# B&R Automation Studio project NAEUL004C00R13L518F00 (part 60)

#### InputRef.var - not listed in the package file held
```iecst
(*2019-03-22*)
(**)
(*General*)
VAR
	p_udiMax : REFERENCE TO UDINT;
	p_udiRstErr : REFERENCE TO UDINT;
END_VAR
(**)
(*Configuration*)
VAR
	p_tyDISettings : REFERENCE TO tyDigitalInputSettings;
	p_sProgNm : REFERENCE TO STRING[15];
END_VAR
(**)
VAR
	p_diConvLftSenOnTm : REFERENCE TO DINT;
	p_diConvLftSenOffTm : REFERENCE TO DINT;
	p_diConvMidSenOnTm : REFERENCE TO DINT;
	p_diConvMidSenOffTm : REFERENCE TO DINT;
	p_diConvRgtSenOnTm : REFERENCE TO DINT;
	p_diConvRgtSenOffTm : REFERENCE TO DINT;
	p_diConvClrSenOnTm : REFERENCE TO DINT;
	p_diConvClrSenOffTm : REFERENCE TO DINT;
	p_diMagConvEntSenOnTm : REFERENCE TO DINT;
	p_diMagConvEntSenOffTm : REFERENCE TO DINT;
	p_diMagConvPresentSenOnTm : REFERENCE TO DINT;
	p_diMagConvPresentSenOffTm : REFERENCE TO DINT;
	p_diConvLineAInletSenOnTm : REFERENCE TO DINT;
	p_diConvLineAInletSenOffTm : REFERENCE TO DINT;
	p_diConvLineBInletSenOnTm : REFERENCE TO DINT;
	p_diConvLineBInletSenOffTm : REFERENCE TO DINT;
	p_diConvUSWidthChkSenOnTm : REFERENCE TO DINT;
	p_diConvUSWidthChkSenOffTm : REFERENCE TO DINT;
	p_tyNtParamCurr : REFERENCE TO tyNtParam;
	p_bMcParamUSWidthChkEn : REFERENCE TO BOOL;
END_VAR
(*Self Test Var*)
VAR
	p_bSelfTest : REFERENCE TO BOOL;
	p_bPshrConvHvBrd : REFERENCE TO BOOL;
	p_tyBufferStat1 : REFERENCE TO tyBffrStat;
	p_tyBufferStat2 : REFERENCE TO tyBffrStat;
	p_tyBufferStat3 : REFERENCE TO tyBffrStat;
	p_tySOTSimulate1 : REFERENCE TO tySOTSigmulateSig;
	p_tySOTSimulate2 : REFERENCE TO tySOTSigmulateSig;
	p_tySOTSimulate3 : REFERENCE TO tySOTSigmulateSig;
	p_bUIAGVSimulationOn : REFERENCE TO BOOL;
	p_tyTagFromMes : REFERENCE TO tyStatFromMES;
	p_tyDO : REFERENCE TO tyDigitalOutput;
	p_eULMag : REFERENCE TO eULMag;
	p_bRstErrSafetyRlyRst : REFERENCE TO BOOL;
	p_bRstCurtainSen : REFERENCE TO BOOL;
END_VAR
(*MagConv On/Off Tm*)
VAR
	p_diInMagConvEntSenOnTm : REFERENCE TO DINT;
	p_diInMagConvEntSenOffTm : REFERENCE TO DINT;
	p_diInMagConvExtSenOnTm : REFERENCE TO DINT;
	p_diInMagConvExtSenOffTm : REFERENCE TO DINT;
	p_diInMagConvMidSenOnTm : REFERENCE TO DINT;
	p_diInMagConvMidSenOffTm : REFERENCE TO DINT;
	p_diOutMagConvEntSenOnTm : REFERENCE TO DINT;
	p_diOutMagConvEntSenOffTm : REFERENCE TO DINT;
	p_diOutMagConvExtSenOnTm : REFERENCE TO DINT;
	p_diOutMagConvExtSenOffTm : REFERENCE TO DINT;
	p_diOutMagConvMidSenOnTm : REFERENCE TO DINT;
	p_diOutMagConvMidSenOffTm : REFERENCE TO DINT;
	p_diInMagConv2EntSenOnTm : REFERENCE TO DINT;
	p_diInMagConv2EntSenOffTm : REFERENCE TO DINT;
	p_diInMagConv2ExtSenOnTm : REFERENCE TO DINT;
	p_diInMagConv2ExtSenOffTm : REFERENCE TO DINT;
	p_diInMagConv2MidSenOnTm : REFERENCE TO DINT;
	p_diInMagConv2MidSenOffTm : REFERENCE TO DINT;
	p_diOutMagConv2EntSenOnTm : REFERENCE TO DINT;
	p_diOutMagConv2EntSenOffTm : REFERENCE TO DINT;
	p_diOutMagConv2ExtSenOnTm : REFERENCE TO DINT;
	p_diOutMagConv2ExtSenOffTm : REFERENCE TO DINT;
	p_diOutMagConv2MidSenOnTm : REFERENCE TO DINT;
	p_diOutMagConv2MidSenOffTm : REFERENCE TO DINT;
	p_bOpsRun : REFERENCE TO BOOL;
	p_bManual : REFERENCE TO BOOL;
	p_bCurtainSenPrep : REFERENCE TO BOOL;
	p_bBypassLifMagInletShute : REFERENCE TO BOOL;
	p_eMidSenNcNoType : REFERENCE TO eMidSenParam;
END_VAR
```

#### InputRef_Link.var - not listed in the package file held
```iecst
(*2019-04-09*)
(**)
(*External Data*)
VAR
	p_eLinkAGVComProtocol : REFERENCE TO eMcAGVCommProtocol;
	p_bLinkNtParamProjSOTSenPrep : REFERENCE TO BOOL;
	p_bLinkStartupRun : REFERENCE TO BOOL;
	p_bOpsTravLifULBypCurtainSenCtrl : REFERENCE TO BOOL;
END_VAR
```

#### Act_Alarm1.st - not listed in the package file held
```iecst
(** 2019-03-25 **)
ACTION Act_Alarm1:

	//Error
	IF EDGEPOS(eStatus1 = Error) THEN

		tyAlmData1.sProgNm		:= p_sProgNm;
		tyAlmData1.udiCode		:= udiStatus1;
		tyAlmData1.eSeverity	:= AlmSeverityError;
		tyAlmData1.udiRunTime	:= tyAlmData1.udiRunTime + 1;
		tyAlmData1.bAlm			:= TRUE;
		tyAlmData1.udiModuleNum  := udiModuleNum;
		g_sDInputProgNm		:= p_sProgNm;

		//Get Error Message
		IF tyAlmData1.udiCode < 10000 OR tyAlmData1.udiCode > 10099 THEN
			tyAlmData1.sAlmMsg	:= 'Unknown';
			tyAlmData1.sRcyMsg	:= 'Unknown';
		ELSE
			tyAlmData1.sAlmMsg	:= a_tyAlmText[tyAlmData1.udiCode].sAlmText;
			tyAlmData1.sRcyMsg	:= a_tyAlmText[tyAlmData1.udiCode].sRcyText;
		END_IF

	ELSIF bRstErr AND (tyAlmData1.udiCode <> 0) THEN

		tyAlmData1.udiCode		:= 0;
		tyAlmData1.eSeverity	:= AlmSeverityNA;
		tyAlmData1.sAlmMsg		:= '';
		tyAlmData1.sRcyMsg		:= '';
		tyAlmData1.bAlm			:= FALSE;
	END_IF

END_ACTION
```

#### Act_Alarm2.st - not listed in the package file held
```iecst
(** 2019-03-25 **)
ACTION Act_Alarm2:

	//Error
	IF EDGEPOS(eStatus2 = Error) THEN

		tyAlmData2.sProgNm		:= p_sProgNm;
		tyAlmData2.udiCode		:= udiStatus2;
		tyAlmData2.eSeverity	:= AlmSeverityError;
		tyAlmData2.udiRunTime	:= tyAlmData2.udiRunTime + 1;
		tyAlmData2.bAlm			:= TRUE;
		tyAlmData2.udiModuleNum  := udiModuleNum;
		g_sDInputProgNm		:= p_sProgNm;
		//Get Error Message
		IF tyAlmData2.udiCode < 10000 OR tyAlmData2.udiCode > 10099 THEN
			tyAlmData2.sAlmMsg	:= 'Unknown';
			tyAlmData2.sRcyMsg	:= 'Unknown';
		ELSE
			tyAlmData2.sAlmMsg	:= a_tyAlmText[tyAlmData2.udiCode].sAlmText;
			tyAlmData2.sRcyMsg	:= a_tyAlmText[tyAlmData2.udiCode].sRcyText;
		END_IF

	ELSIF bRstErr AND (tyAlmData2.udiCode <> 0) THEN

		tyAlmData2.udiCode		:= 0;
		tyAlmData2.eSeverity	:= AlmSeverityNA;
		tyAlmData2.sAlmMsg		:= '';
		tyAlmData2.sRcyMsg		:= '';
		tyAlmData2.bAlm			:= FALSE;
	END_IF

END_ACTION
```

#### Act_Alarm3.st - not listed in the package file held
```iecst
(** 2019-03-25 **)
ACTION Act_Alarm3:

	//Error
	IF EDGEPOS(eStatus3 = Error) THEN

		tyAlmData3.sProgNm		:= p_sProgNm;
		tyAlmData3.udiCode		:= udiStatus3;
		tyAlmData3.eSeverity	:= AlmSeverityError;
		tyAlmData3.udiRunTime	:= tyAlmData3.udiRunTime + 1;
		tyAlmData3.bAlm			:= TRUE;
		tyAlmData3.udiModuleNum  := udiModuleNum;
		g_sDInputProgNm		:= p_sProgNm;
		//Get Error Message
		IF tyAlmData3.udiCode < 10000 OR tyAlmData3.udiCode > 10099 THEN
			tyAlmData3.sAlmMsg	:= 'Unknown';
			tyAlmData3.sRcyMsg	:= 'Unknown';
		ELSE
			tyAlmData3.sAlmMsg	:= a_tyAlmText[tyAlmData3.udiCode].sAlmText;
			tyAlmData3.sRcyMsg	:= a_tyAlmText[tyAlmData3.udiCode].sRcyText;
		END_IF

	ELSIF bRstErr AND (tyAlmData3.udiCode <> 0) THEN

		tyAlmData3.udiCode		:= 0;
		tyAlmData3.eSeverity	:= AlmSeverityNA;
		tyAlmData3.sAlmMsg		:= '';
		tyAlmData3.sRcyMsg		:= '';
		tyAlmData3.bAlm			:= FALSE;
	END_IF

END_ACTION
```

#### Act_Alarm4.st - not listed in the package file held
```iecst
(** 2019-03-25 **)
ACTION Act_Alarm4:

	//Error
	IF EDGEPOS(eStatus4 = Error) THEN

		tyAlmData4.sProgNm		:= p_sProgNm;
		tyAlmData4.udiCode		:= udiStatus4;
		tyAlmData4.eSeverity	:= AlmSeverityError;
		tyAlmData4.udiRunTime	:= tyAlmData4.udiRunTime + 1;
		tyAlmData4.bAlm			:= TRUE;
		tyAlmData4.udiModuleNum  := udiModuleNum;
		g_sDInputProgNm		:= p_sProgNm;
		//Get Error Message
		IF tyAlmData4.udiCode < 10000 OR tyAlmData4.udiCode > 10099 THEN
			tyAlmData4.sAlmMsg	:= 'Unknown';
			tyAlmData4.sRcyMsg	:= 'Unknown';
		ELSE
			tyAlmData4.sAlmMsg	:= a_tyAlmText[tyAlmData4.udiCode].sAlmText;
			tyAlmData4.sRcyMsg	:= a_tyAlmText[tyAlmData4.udiCode].sRcyText;
		END_IF

	ELSIF bRstErr AND (tyAlmData4.udiCode <> 0) THEN

		tyAlmData4.udiCode		:= 0;
		tyAlmData4.eSeverity	:= AlmSeverityNA;
		tyAlmData4.sAlmMsg		:= '';
		tyAlmData4.sRcyMsg		:= '';
		tyAlmData4.bAlm			:= FALSE;
	END_IF

END_ACTION
```

#### Act_Alarm5.st - not listed in the package file held
```iecst
(** 2019-03-25 **)
ACTION Act_Alarm5:

	//Error
	IF EDGEPOS(eStatus5 = Error) THEN

		tyAlmData5.sProgNm		:= p_sProgNm;
		tyAlmData5.udiCode		:= udiStatus5;
		tyAlmData5.eSeverity	:= AlmSeverityError;
		tyAlmData5.udiRunTime	:= tyAlmData5.udiRunTime + 1;
		tyAlmData5.bAlm			:= TRUE;
		tyAlmData5.udiModuleNum  := udiModuleNum;
		g_sDInputProgNm		:= p_sProgNm;
		//Get Error Message
		IF tyAlmData5.udiCode < 10000 OR tyAlmData5.udiCode > 10099 THEN
			tyAlmData5.sAlmMsg	:= 'Unknown';
			tyAlmData5.sRcyMsg	:= 'Unknown';
		ELSE
			tyAlmData5.sAlmMsg	:= a_tyAlmText[tyAlmData5.udiCode].sAlmText;
			tyAlmData5.sRcyMsg	:= a_tyAlmText[tyAlmData5.udiCode].sRcyText;
		END_IF

	ELSIF bRstErr AND (tyAlmData5.udiCode <> 0) THEN

		tyAlmData5.udiCode		:= 0;
		tyAlmData5.eSeverity	:= AlmSeverityNA;
		tyAlmData5.sAlmMsg		:= '';
		tyAlmData5.sRcyMsg		:= '';
		tyAlmData5.bAlm			:= FALSE;
	END_IF

END_ACTION
```

#### Act_Alarm6.st - not listed in the package file held
```iecst
(** 2019-03-25 **)
ACTION Act_Alarm6:

	//Error
	IF EDGEPOS(eStatus6 = Error) THEN

		tyAlmData6.sProgNm		:= p_sProgNm;
		tyAlmData6.udiCode		:= udiStatus6;
		tyAlmData6.eSeverity	:= AlmSeverityError;
		tyAlmData6.udiRunTime	:= tyAlmData6.udiRunTime + 1;
		tyAlmData6.bAlm			:= TRUE;
		tyAlmData6.udiModuleNum  := udiModuleNum;
		g_sDInputProgNm		:= p_sProgNm;
		//Get Error Message
		IF tyAlmData6.udiCode < 10000 OR tyAlmData6.udiCode > 10099 THEN
			tyAlmData6.sAlmMsg	:= 'Unknown';
			tyAlmData6.sRcyMsg	:= 'Unknown';
		ELSE
			tyAlmData6.sAlmMsg	:= a_tyAlmText[tyAlmData6.udiCode].sAlmText;
			tyAlmData6.sRcyMsg	:= a_tyAlmText[tyAlmData6.udiCode].sRcyText;
		END_IF

	ELSIF bRstErr AND (tyAlmData6.udiCode <> 0) THEN

		tyAlmData6.udiCode		:= 0;
		tyAlmData6.eSeverity	:= AlmSeverityNA;
		tyAlmData6.sAlmMsg		:= '';
		tyAlmData6.sRcyMsg		:= '';
		tyAlmData6.bAlm			:= FALSE;
	END_IF

END_ACTION
```

#### Act_InitGlobal.st - not listed in the package file held
```iecst
(** 2018-12-10 **)
ACTION Act_InitGlobal:

	(* Always Change If Project Change *)

	//Pass Data To Link
	p_eLinkAGVComProtocol ACCESS p_McParamAGVComProtocol;
	p_bLinkNtParamProjSOTSenPrep ACCESS p_NtParamProjSOTSenPrep;
	p_bLinkStartupRun ACCESS p_StartupRun;
	p_bOpsTravLifULBypCurtainSenCtrl ACCESS p_OpsTravLifULBypCurtainSenCtrl;
	p_bOpsRun ACCESS p_OpsRun;
	p_bCurtainSenPrep ACCESS p_NtParamCurtainSenPrep;

	//Pass Data To Internal Use
	p_udiRstErr ACCESS p_RstErrReset;
	p_tyDISettings ACCESS p_NtParamDISettings;
	p_sProgNm ACCESS p_NtParamDIProgNm;

	p_diConvLftSenOnTm ACCESS p_McParamConvLftSenOnTm;
	p_diConvLftSenOffTm ACCESS p_McParamConvLftSenOffTm;
	p_diConvMidSenOnTm ACCESS p_McParamConvMidSenOnTm;
	p_diConvMidSenOffTm ACCESS p_McParamConvMidSenOffTm;
	p_diConvRgtSenOnTm ACCESS p_McParamConvRgtSenOnTm;
	p_diConvRgtSenOffTm ACCESS p_McParamConvRgtSenOffTm;
	p_diConvClrSenOnTm ACCESS p_McParamConvClrSenOnTm;
	p_diConvClrSenOffTm ACCESS p_McParamConvClrSenOffTm;

	p_diMagConvEntSenOnTm ACCESS p_McParamMagConvEntrySenOnTm;
	p_diMagConvEntSenOffTm ACCESS p_McParamMagConvEntrySenOffTm;
	p_diMagConvPresentSenOnTm ACCESS p_McParamMagConvPresentSenOnTm;
	p_diMagConvPresentSenOffTm ACCESS p_McParamMagConvPresentSenOffTm;

	p_tyBufferStat1 ACCESS p_Buffer1BffrStat;
	p_tyBufferStat2 ACCESS p_Buffer2BffrStat;
	p_tyBufferStat3 ACCESS p_Buffer3BffrStat;
	p_bSelfTest ACCESS p_OpsTravLifULSelfTest;
	p_bPshrConvHvBrd ACCESS p_PshrConvHvBrd;

	p_bUIAGVSimulationOn ACCESS p_UIAGVSimulationOn;
	p_tySOTSimulate1 ACCESS p_UISOTSimulationSig1;
	p_tySOTSimulate2 ACCESS p_UISOTSimulationSig2;
	p_tySOTSimulate3 ACCESS p_UISOTSimulationSig3;

	p_tyTagFromMes ACCESS p_TagFromMes;
	p_tyDO  ACCESS p_DO;
	p_eULMag ACCESS p_NtParamProjMag;
	p_bRstErrSafetyRlyRst ACCESS p_RstErrSafetyRlyRst;

	p_diConvLineAInletSenOnTm ACCESS p_McParamConvLineAInletSenOnTm;
	p_diConvLineAInletSenOffTm ACCESS p_McParamConvLineAInletSenOffTm;
	p_diConvLineBInletSenOnTm ACCESS p_McParamConvLineBInletSenOnTm;
	p_diConvLineBInletSenOffTm ACCESS p_McParamConvLineBInletSenOffTm;
	p_diConvUSWidthChkSenOnTm ACCESS p_McParamUSWidthChkSenOnTm;
	p_diConvUSWidthChkSenOffTm ACCESS p_McParamUSWidthChkSenOffTm;

	p_tyNtParamCurr ACCESS p_NtParamCurr;
	p_bMcParamUSWidthChkEn ACCESS p_McParamUSWidthChkEn;

	//MagConv IN/OUT
	p_diInMagConvEntSenOnTm ACCESS p_McParamInMagConvEntSenOnTm;
	p_diInMagConvEntSenOffTm ACCESS p_McParamInMagConvEntSenOffTm;
	p_diInMagConvExtSenOnTm ACCESS p_McParamInMagConvExtSenOnTm;
	p_diInMagConvExtSenOffTm ACCESS p_McParamInMagConvExtSenOffTm;
	p_diInMagConvMidSenOnTm ACCESS p_McParamInMagConvMidSenOnTm;
	p_diInMagConvMidSenOffTm ACCESS p_McParamInMagConvMidSenOffTm;

	p_diOutMagConvEntSenOnTm ACCESS p_McParamOutMagConvEntSenOnTm;
	p_diOutMagConvEntSenOffTm ACCESS p_McParamOutMagConvEntSenOffTm;
	p_diOutMagConvExtSenOnTm ACCESS p_McParamOutMagConvExtSenOnTm;
	p_diOutMagConvExtSenOffTm ACCESS p_McParamOutMagConvExtSenOffTm;
	p_diOutMagConvMidSenOnTm ACCESS p_McParamOutMagConvMidSenOnTm;
	p_diOutMagConvMidSenOffTm ACCESS p_McParamOutMagConvMidSenOffTm;

	p_diInMagConv2EntSenOnTm ACCESS p_McParamInMagConv2EntSenOnTm;
	p_diInMagConv2EntSenOffTm ACCESS p_McParamInMagConv2EntSenOffTm;
	p_diInMagConv2ExtSenOnTm ACCESS p_McParamInMagConv2ExtSenOnTm;
	p_diInMagConv2ExtSenOffTm ACCESS p_McParamInMagConv2ExtSenOffTm;
	p_diInMagConv2MidSenOnTm ACCESS p_McParamInMagConv2MidSenOnTm;
	p_diInMagConv2MidSenOffTm ACCESS p_McParamInMagConv2MidSenOffTm;

	p_diOutMagConv2EntSenOnTm ACCESS p_McParamOutMagConv2EntSenOnTm;
	p_diOutMagConv2EntSenOffTm ACCESS p_McParamOutMagConv2EntSenOffTm;
	p_diOutMagConv2ExtSenOnTm ACCESS p_McParamOutMagConv2ExtSenOnTm;
	p_diOutMagConv2ExtSenOffTm ACCESS p_McParamOutMagConv2ExtSenOffTm;
	p_diOutMagConv2MidSenOnTm ACCESS p_McParamOutMagConv2MidSenOnTm;
	p_diOutMagConv2MidSenOffTm ACCESS p_McParamOutMagConv2MidSenOffTm;

	p_bRstCurtainSen ACCESS p_UISafetyCurtainReset;
	p_bManual ACCESS p_UIMnlMod;

	p_eMidSenNcNoType ACCESS p_NtParamMidSenNcNo;

	(* Always Change If Project Change *)

END_ACTION
```

#### Act_InitLocal.st - not listed in the package file held
```iecst
(** 2019-03-25 **)
ACTION Act_InitLocal:

	//Input Reference Link To Local Variable
	p_udiMax ACCESS ADR(c_udiDInputMax);
	p_udiRstErr ACCESS ADR(udiRstErr);
	p_tyDISettings ACCESS ADR(tyDISettings);
	p_sProgNm ACCESS ADR(sProgNm);

	p_diConvLftSenOnTm ACCESS ADR(diConvLftSenOnTm);
	p_diConvLftSenOffTm ACCESS ADR(diConvLftSenOffTm);
	p_diConvMidSenOnTm ACCESS ADR(diConvMidSenOnTm);
	p_diConvMidSenOffTm ACCESS ADR(diConvMidSenOffTm);
	p_diConvRgtSenOnTm ACCESS ADR(diConvRgtSenOnTm);
	p_diConvRgtSenOffTm ACCESS ADR(diConvRgtSenOffTm);
	p_diConvClrSenOnTm ACCESS ADR(diConvClrSenOnTm);
	p_diConvClrSenOffTm ACCESS ADR(diConvClrSenOffTm);
	p_diMagConvEntSenOnTm ACCESS ADR(diMagConvEntSenOnTm);
	p_diMagConvEntSenOffTm ACCESS ADR(diMagConvEntSenOffTm);
	p_diMagConvPresentSenOnTm ACCESS ADR(diMagConvPresentSenOnTm);
	p_diMagConvPresentSenOffTm ACCESS ADR(diMagConvPresentSenOffTm);

	//MagConv IN/OUT
	p_diInMagConvEntSenOnTm ACCESS ADR(diInMagConvEntSenOnTm);
	p_diInMagConvEntSenOffTm ACCESS ADR(diInMagConvEntSenOffTm);
	p_diInMagConvExtSenOnTm ACCESS ADR(diInMagConvExtSenOnTm);
	p_diInMagConvExtSenOffTm ACCESS ADR(diInMagConvExtSenOffTm);
	p_diInMagConvMidSenOnTm ACCESS ADR(diInMagConvMidSenOnTm);
	p_diInMagConvMidSenOffTm ACCESS ADR(diInMagConvMidSenOffTm);

	p_diOutMagConvEntSenOnTm ACCESS ADR(diOutMagConvEntSenOnTm);
	p_diOutMagConvEntSenOffTm ACCESS ADR(diOutMagConvEntSenOffTm);
	p_diOutMagConvExtSenOnTm ACCESS ADR(diOutMagConvExtSenOnTm);
	p_diOutMagConvExtSenOffTm ACCESS ADR(diOutMagConvExtSenOffTm);
	p_diOutMagConvMidSenOnTm ACCESS ADR(diOutMagConvMidSenOnTm);
	p_diOutMagConvMidSenOffTm ACCESS ADR(diOutMagConvMidSenOffTm);

	p_diInMagConv2EntSenOnTm ACCESS ADR(diInMagConv2EntSenOnTm);
	p_diInMagConv2EntSenOffTm ACCESS ADR(diInMagConv2EntSenOffTm);
	p_diInMagConv2ExtSenOnTm ACCESS ADR(diInMagConv2ExtSenOnTm);
	p_diInMagConv2ExtSenOffTm ACCESS ADR(diInMagConv2ExtSenOffTm);
	p_diInMagConv2MidSenOnTm ACCESS ADR(diInMagConv2MidSenOnTm);
	p_diInMagConv2MidSenOffTm ACCESS ADR(diInMagConv2MidSenOffTm);

	p_diOutMagConv2EntSenOnTm ACCESS ADR(diOutMagConv2EntSenOnTm);
	p_diOutMagConv2EntSenOffTm ACCESS ADR(diOutMagConv2EntSenOffTm);
	p_diOutMagConv2ExtSenOnTm ACCESS ADR(diOutMagConv2ExtSenOnTm);
	p_diOutMagConv2ExtSenOffTm ACCESS ADR(diOutMagConv2ExtSenOffTm);
	p_diOutMagConv2MidSenOnTm ACCESS ADR(diOutMagConv2MidSenOnTm);
	p_diOutMagConv2MidSenOffTm ACCESS ADR(diOutMagConv2MidSenOffTm);

//	p_eMidSenNcNoType		ACCESS ADR(eMidSenNcNoType);
END_ACTION
```

#### Act_Link.st - not listed in the package file held
```iecst
(** 2021-08-04 **)
ACTION Act_Link:

END_ACTION
```

#### Init.st - not listed in the package file held
```iecst
(** 2019-03-22 **)
PROGRAM _INIT

	(* Always Change If Project Change *)

	//Pass Address To Global Address For External Use
	//Action, State & Status

	//Alarm
	p_DIAlmData1	:= ADR(tyAlmData1);
	p_DIAlmData2	:= ADR(tyAlmData2);
	p_DIAlmData3	:= ADR(tyAlmData3);
	p_DIAlmData4	:= ADR(tyAlmData4);
	p_DIAlmData5	:= ADR(tyAlmData5);
	p_DIAlmData6    := ADR(tyAlmData6);

	//Output
	p_DI					:= ADR(tyDInput);
	p_DISafetyRlySig		:= ADR(tyDInput.bSafetyRlySig);
	p_DIEStopSig			:= ADR(tyDInput.bEStopSig);
	p_DICoverSWSig			:= ADR(tyDInput.bCoverSWSig);
	p_DIUBAA				:= ADR(tyDInput.bUBAA);
	p_DIUBAB				:= ADR(tyDInput.bUBAB);
	p_DIUBAAStat			:= ADR(tyDInput.bUBAAStat);
	p_DIUBABStat			:= ADR(tyDInput.bUBABStat);
	p_DIPusherExtRS			:= ADR(tyDInput.bPusherExtRS);
	p_DIPusherRetRS			:= ADR(tyDInput.bPusherRetRS);
	p_DIConvLftSen			:= ADR(tyDInput.bConvLftSen);
	p_DIConvMidSen			:= ADR(tyDInput.bConvMidSen);
	p_DIConvRgtSen			:= ADR(tyDInput.bConvRgtSen);
	p_DIConvClrSen			:= ADR(tyDInput.bConvClrSen);
	p_DIOvenInfeedSigA		:= ADR(tyDInput.bOvenInfeedSigA);
	p_DIOvenInfeedSigB		:= ADR(tyDInput.bOvenInfeedSigB);
	p_DILifterTimingBeltSen	:= ADR(tyDInput.bLifterTimingBeltSen);
	p_DILifterSafetyLmtSW1	:= ADR(tyDInput.bLifterSafetyLmtSW1);
	p_DILifterSafetyLmtSW2	:= ADR(tyDInput.bLifterSafetyLmtSW2);
	p_DIMag1FixedClampRS	:= ADR(tyDInput.bMag1FixedClampRS);
	p_DIMag1FixedUnclampRS	:= ADR(tyDInput.bMag1FixedUnclampRS);
	p_DIMag1RemoteClampRS	:= ADR(tyDInput.bMag1RemoteClampRS);
	p_DIMag1RemoteUnclampRS := ADR(tyDInput.bMag1RemoteUnclampRS);
	p_DIMag2FixedClampRS	:= ADR(tyDInput.bMag2FixedClampRS);
	p_DIMag2FixedUnclampRS	:= ADR(tyDInput.bMag2FixedUnclampRS);
	p_DIMag2RemoteClampRS	:= ADR(tyDInput.bMag2RemoteClampRS);
	p_DIMag2RemoteUnclampRS	:= ADR(tyDInput.bMag2RemoteUnclampRS);
	p_DIMag3FixedClampRS	:= ADR(tyDInput.bMag3FixedClampRS);
	p_DIMag3FixedUnclampRS	:= ADR(tyDInput.bMag3FixedUnclampRS);
	p_DIMag3RemoteClampRS	:= ADR(tyDInput.bMag3RemoteClampRS);
	p_DIMag3RemoteUnclampRS	:= ADR(tyDInput.bMag3RemoteUnclampRS);
	p_DIInShutterOpenRS		:= ADR(tyDInput.bInShutterOpenRS);
	p_DIInShutterCloseRS	:= ADR(tyDInput.bInShutterCloseRS);
	p_DIOutShutterOpenRS	:= ADR(tyDInput.bOutShutterOpenRS);
	p_DIOutShutterCloseRS	:= ADR(tyDInput.bOutShutterCloseRS);
	p_DIMagPresentSen1		:= ADR(tyDInput.bMagPresentSen1);
	p_DIMagPresentSen2		:= ADR(tyDInput.bMagPresentSen2);
	p_DIMagPresentSen3		:= ADR(tyDInput.bMagPresentSen3);
	p_DIMagConvEntSen1		:= ADR(tyDInput.bMagConvEntSen1);
	p_DIMagConvEntSen2		:= ADR(tyDInput.bMagConvEntSen2);
	p_DIMagConvEntSen3		:= ADR(tyDInput.bMagConvEntSen3);
	p_DIMag1AIVInPosSen1	:= ADR(tyDInput.bMag1AIVInPosSen1);
	p_DIMag1AIVInPosSen2	:= ADR(tyDInput.bMag1AIVInPosSen2);
	p_DIMag2AIVInPosSen1	:= ADR(tyDInput.bMag2AIVInPosSen1);
	p_DIMag2AIVInPosSen2	:= ADR(tyDInput.bMag2AIVInPosSen2);
	p_DIMag3AIVInPosSen1	:= ADR(tyDInput.bMag3AIVInPosSen1);
	p_DIMag3AIVInPosSen2	:= ADR(tyDInput.bMag3AIVInPosSen2);
	p_DIMag1OrientChkSen1	:= ADR(tyDInput.bMag1OrientChkSen1);
	p_DIMag1OrientChkSen2	:= ADR(tyDInput.bMag1OrientChkSen2);
	p_DIMag2OrientChkSen1	:= ADR(tyDInput.bMag2OrientChkSen1);
	p_DIMag2OrientChkSen2	:= ADR(tyDInput.bMag2OrientChkSen2);
	p_DIMag3OrientChkSen1	:= ADR(tyDInput.bMag3OrientChkSen1);
	p_DIMag3OrientChkSen2	:= ADR(tyDInput.bMag3OrientChkSen2);
	p_DIUSWidthChkSen		:= ADR(tyDInput.bUSWidthChkSen);
	p_DIMagConvHeightSen1	:= ADR(tyDInput.bMagConvHeightSen1);
	p_DIMagConvHeightSen2	:= ADR(tyDInput.bMagConvHeightSen2);
	p_DIMagConvHeightSen3	:= ADR(tyDInput.bMagConvHeightSen3);
	p_DIMagConvSmallMagSen1	:= ADR(tyDInput.bMagConvSmallMagSen1);
	p_DIMagConvSmallMagSen2	:= ADR(tyDInput.bMagConvSmallMagSen2);
	p_DIMagConvSmallMagSen3	:= ADR(tyDInput.bMagConvSmallMagSen3);
	p_DIMagConvLargeMagSen1	:= ADR(tyDInput.bMagConvLargeMagSen1);
	p_DIMagConvLargeMagSen2	:= ADR(tyDInput.bMagConvLargeMagSen2);
	p_DIMagConvLargeMagSen3	:= ADR(tyDInput.bMagConvLargeMagSen3);
	p_DIMagConvCAB717MagSen1:= ADR(tyDInput.bMagConvCAB717MagSen1);
	p_DIMagConvCAB717MagSen2:= ADR(tyDInput.bMagConvCAB717MagSen2);
	p_DIMagConvCAB717MagSen3:= ADR(tyDInput.bMagConvCAB717MagSen3);
	p_DIMag1SelUnclampRS	:= ADR(tyDInput.bMag1SelUnClampRS);
	p_DIMag2SelUnclampRS	:= ADR(tyDInput.bMag2SelUnClampRS);
	p_DIMag3SelUnclampRS	:= ADR(tyDInput.bMag3SelUnClampRS);
	p_DIMag1SafetyBarExtRS	:= ADR(tyDInput.bMag1SafetyBarExtRS);
	p_DIMag1SafetyBarRetRS	:= ADR(tyDInput.bMag1SafetyBarRetRS);
	p_DIMag2SafetyBarExtRS	:= ADR(tyDInput.bMag2SafetyBarExtRS);
	p_DIMag2SafetyBarRetRS	:= ADR(tyDInput.bMag2SafetyBarRetRS);
	p_DIMag3SafetyBarExtRS	:= ADR(tyDInput.bMag3SafetyBarExtRS);
	p_DIMag3SafetyBarRetRS	:= ADR(tyDInput.bMag3SafetyBarRetRS);
	p_DIMag1WallEngageRS	:= ADR(tyDInput.bMag1WallEngageRS);
	p_DIMag1WallDisengageRS	:= ADR(tyDInput.bMag1WallDisengageRS);
	p_DIMag2WallEngageRS	:= ADR(tyDInput.bMag2WallEngageRS);
	p_DIMag2WallDisengageRS	:= ADR(tyDInput.bMag2WallDisengageRS);
	p_DIMag3WallEngageRS	:= ADR(tyDInput.bMag3WallEngageRS);
	p_DIMag3WallDisengageRS	:= ADR(tyDInput.bMag3WallDisengageRS);
	p_DISOT1Receive 		:= ADR(tyDInput.bSOT1Receive);
	p_DISOT1Error 			:= ADR(tyDInput.bSOT1AIVError);
	p_DISOT1SizeLarge		:= ADR(tyDInput.bSOT1AIVSizeLarge);
	p_DISOT1Ready			:= ADR(tyDInput.bSOT1AIVReady);
	p_DISOT1Available		:= ADR(tyDInput.bSOT1AIVAvailable);
	p_DISOT2Receive 		:= ADR(tyDInput.bSOT2Receive);
	p_DISOT2Error 			:= ADR(tyDInput.bSOT2AIVError);
	p_DISOT2SizeLarge		:= ADR(tyDInput.bSOT2AIVSizeLarge);
	p_DISOT2Ready			:= ADR(tyDInput.bSOT2AIVReady);
	p_DISOT2Available		:= ADR(tyDInput.bSOT2AIVAvailable);
	p_DISOT3Receive 		:= ADR(tyDInput.bSOT3Receive);
	p_DISOT3Error 			:= ADR(tyDInput.bSOT3AIVError);
	p_DISOT3SizeLarge		:= ADR(tyDInput.bSOT3AIVSizeLarge);
	p_DISOT3Ready			:= ADR(tyDInput.bSOT3AIVReady);
	p_DISOT3Available		:= ADR(tyDInput.bSOT3AIVAvailable);
	p_DIFleetManagerActive  := ADR(tyDInput.bFleetManagerReady);
	p_DIPusherExtSlwSen		:= ADR(tyDInput.bPusherExtSlwSen);
	p_DIPusherRetSlwSen		:= ADR(tyDInput.bPusherRetSlwSen);
	p_DIMtrPshrTorqueSig	:= ADR(tyDInput.bMtrPshrTorqueSig);
	p_DIMtrPshrAlmSig		:= ADR(tyDInput.bMtrPshrAlmSig);
	p_DIMagWidthChkSen		:= ADR(tyDInput.bMagWidthChkSen);
	p_DIUSWidthChkSen		:= ADR(tyDInput.bUSWidthChkSen);
	p_DIConvLineAInletSen	:= ADR(tyDInput.bConvLineAInletSen);
	p_DIConvLineBInletSen	:= ADR(tyDInput.bConvLineBInletSen);
	p_DIPshrAntiJamSen		:= ADR(tyDInput.bPshrAntiJam);

	p_DIInMagConvEntSen		:= ADR(tyDInput.bInMagConvEntSen);
	p_DIInMagConvMidSen		:= ADR(tyDInput.bInMagConvMidSen);
	p_DIInMagConvExtSen		:= ADR(tyDInput.bInMagConvExtSen);
	p_DIOutMagConvEntSen	:= ADR(tyDInput.bOutMagConvEntSen);
	p_DIOutMagConvMidSen	:= ADR(tyDInput.bOutMagConvMidSen);
	p_DIOutMagConvExtSen	:= ADR(tyDInput.bOutMagConvExtSen);
	p_DIInMagConv2EntSen	:= ADR(tyDInput.bInMagConv2EntSen);
	p_DIInMagConv2MidSen	:= ADR(tyDInput.bInMagConv2MidSen);
	p_DIInMagConv2ExtSen	:= ADR(tyDInput.bInMagConv2ExtSen);
	p_DIOutMagConv2EntSen	:= ADR(tyDInput.bOutMagConv2EntSen);
	p_DIOutMagConv2MidSen	:= ADR(tyDInput.bOutMagConv2MidSen);
	p_DIOutMagConv2ExtSen	:= ADR(tyDInput.bOutMagConv2ExtSen);
	p_DILifterLmtSW			:= ADR(tyDInput.bLifterLmtSW); //~~PresentSen1
	p_DILifter2LmtSW		:= ADR(tyDInput.bLifter2LmtSW);//~~PresentSen2
	p_DIMtrOverloadSig		:= ADR(tyDInput.bMtrOverloadSig);

	p_DIOutShutterOpenRS2	:= ADR(tyDInput.bOutShutterOpenRS2);
	p_DIOutShutterCloseRS2	:= ADR(tyDInput.bOutShutterCloseRS2);

	p_DIOutShutterOpenRS3	:= ADR(tyDInput.bOutShutterOpenRS3);
	p_DIOutShutterCloseRS3	:= ADR(tyDInput.bOutShutterCloseRS3);

	p_DIMag1FixedClampSen	:= ADR(tyDInput.bMag1FixedClampSen);
	p_DIMag2FixedClampSen	:= ADR(tyDInput.bMag2FixedClampSen);
	p_DIMag3FixedClampSen	:= ADR(tyDInput.bMag3FixedClampSen);

	p_DICurtainSen			:= ADR(tyDInput.bCurtainSen);
	p_DICurtainSenPB		:= ADR(tyDInput.bCurtainSenPB);

	p_DIHighMagDetSen1		:= ADR(tyDInput.bHighMagDetSen1); // Detect the Magazine Height together with magazine orientation
	p_DIHighMagDetSen2		:= ADR(tyDInput.bHighMagDetSen2);
	p_DIHighMagDetSen3		:= ADR(tyDInput.bHighMagDetSen3);															//as mag orientation sen is always detecting magazine at any orientation
	//For magazine without metal plate detecting
	p_DIInletStopperASen	:= ADR(tyDInput.bInletStopperASen);
	p_DIPCBScanComplSig		:= ADR(tyDInput.diScanComplSig);

	p_DILifterSafetyStatus		:= ADR(eStatus4);
	(* Always Change If Project Change *)

END_PROGRAM
```

### DOutput.typ - Change By Project
```iecst
(*2018-12-13*)
(**)
(*Action*)

TYPE
	eDOAction :
		(
		DOActIdle,
		DOActRstAll,
		DOActSetBypassCoverSwitch,
		DOActRstBypassCoverSwitch
		);
END_TYPE

(**)
(*Data*)

TYPE
	tyDigitalOutput : 	STRUCT
		bSafetyRlyRst : BOOL;
		bTLRed : BOOL;
		bTLAmber : BOOL;
		bTLGreen : BOOL;
		bBuzzer : BOOL;
		bUSBA : BOOL;
		bUSBB : BOOL;
		bOvenInfoSigA : BOOL;
		bOvenInfoSigB : BOOL;
		bPusherExtCtrl : BOOL;
		bStopperUnBlkCtrlA : BOOL;
		bStopperUnBlkCtrlB : BOOL;
		bMag1FixedClampCtrl : BOOL;
		bMag1RemoteClampCtrl : BOOL;
		bMag2FixedClampCtrl : BOOL;
		bMag2RemoteClampCtrl : BOOL;
		bMag3FixedClampCtrl : BOOL;
		bMag3RemoteClampCtrl : BOOL;
		bInShutterOpenCtrl : BOOL;
		bInShutterCloseCtrl : BOOL;
		bOutShutterOpenCtrl : BOOL;
		bOutShutterCloseCtrl : BOOL;
		bMag1ConvMtrIn : BOOL; (*LifterMagConv*)
		bMag1ConvMtrOut : BOOL;
		bMag2ConvMtrIn : BOOL;
		bMag2ConvMtrOut : BOOL;
		bMag3ConvMtrIn : BOOL;
		bMag3ConvMtrOut : BOOL;
		bMag1SelClampCtrl : BOOL;
		bMag2SelClampCtrl : BOOL;
		bMag3SelClampCtrl : BOOL;
		bPusherConvMtrOn : BOOL;
		bMag1WallEngageCtrl : BOOL;
		bMag2WallEngageCtrl : BOOL;
		bMag3WallEngageCtrl : BOOL;
		bMag1SafetyBarRetCtrl : BOOL;
		bMag2SafetyBarRetCtrl : BOOL;
		bMag3SafetyBarRetCtrl : BOOL;
		bSOT1MagError : BOOL;
		bSOT1MagSizeLarge : BOOL;
		bSOT1MagReady : BOOL;
		bSOT1MagAvailable : BOOL;
		bSOT2MagError : BOOL;
		bSOT2MagSizeLarge : BOOL;
		bSOT2MagReady : BOOL;
		bSOT2MagAvailable : BOOL;
		bSOT3MagError : BOOL;
		bSOT3MagSizeLarge : BOOL;
		bSOT3MagReady : BOOL;
		bSOT3MagAvailable : BOOL;
		bSOT4MagError : BOOL;
		bSOT4MagSizeLarge : BOOL;
		bSOT4MagReady : BOOL;
		bSOT4MagAvailable : BOOL;
		bMagAWOpenLimByp1 : BOOL;
		bMagAWOpenLimByp2 : BOOL;
		bMagAWOpenLimByp3 : BOOL;
		bMagAWOpenLimByp4 : BOOL;
		bMagAWSmallLimSen1 : BOOL;
		bMagAWSmallLimSen2 : BOOL;
		bMagAWSmallLimSen3 : BOOL;
		bMagAWSmallLimSen4 : BOOL;
		bMag1ReqToBring : BOOL;
		bMag1ReqToGet : BOOL;
		bMag2ReqToBring : BOOL;
		bMag2ReqToGet : BOOL;
		bMag3ReqToBring : BOOL;
		bMag3ReqToGet : BOOL;
		bMag4ReqToBring : BOOL;
		bMag4ReqToGet : BOOL;
		bMtrPshrExt : BOOL;
		bMtrPshrRet : BOOL;
		bMtrPshrOn : BOOL;
		bMtrPshrBrakeRls : BOOL;
		bMtrPshrSpdBinBit0 : BOOL;
		bMtrPshrSpdBinBit1 : BOOL;
		bMtrPshrSpdBinBit2 : BOOL;
		bMtrPshrAlmRst : BOOL;
		bInMagConvMtrOn : BOOL;
		bOutMagConvMtrOn : BOOL;
		bInMagConv2MtrOn : BOOL;
		bOutMagConv2MtrOn : BOOL;
		bEntTopStprUnblkCtrl : BOOL; (*MagConv_Top*)
		bMidTopStprUnblkCtrl : BOOL;
		bExtTopStprUnblkCtrl : BOOL;
		bMidBtmStprUnblkCtrl : BOOL;
		bExtBtmStprUnblkCtrl : BOOL;
		bEntTopStprUnblkCtrl2 : BOOL; (*MagConv2_Top*)
		bMidTopStprUnblkCtrl2 : BOOL;
		bExtTopStprUnblkCtrl2 : BOOL;
		bMidBtmStprUnblkCtrl2 : BOOL;
		bExtBtmStprUnblkCtrl2 : BOOL;
		bMtrPwrRly : BOOL;
		bMag1FixedClampOpenCtrl : BOOL;
		bMag1RemoteClampOpenCtrl : BOOL;
		bMag2FixedClampOpenCtrl : BOOL;
		bMag2RemoteClampOpenCtrl : BOOL;
		bMag3FixedClampOpenCtrl : BOOL;
		bMag3RemoteClampOpenCtrl : BOOL;
		bOutShutterOpenCtrl2 : BOOL;
		bOutShutterCloseCtrl2 : BOOL;
		bOutShutterOpenCtrl3 : BOOL;
		bOutShutterCloseCtrl3 : BOOL;
		bBypCurtainSen : BOOL;
		bRstCurtainSen : BOOL;
		bBypCurtainPBLED : BOOL;
		diInletStopperRetCtrl : BOOL;
		diInletStopperExtCtrl : BOOL;
		diScanTrigSig : BOOL;
		diMag1ExitPCB : BOOL;
		diMag2ExitPCB : BOOL;
		diMag3ExitPCB : BOOL;
		bMag1SelUnClampCtrl : BOOL;
	END_STRUCT;
	tyDigitalOutputSettings : 	STRUCT
		diSafetyRlyRst : DINT;
		diTLRed : DINT;
		diTLAmber : DINT;
		diTLGreen : DINT;
		diBuzzer : DINT;
		diUSBA : DINT;
		diUSBB : DINT;
		diOvenInfoSigA : DINT;
		diOvenInfoSigB : DINT;
		diPusherExtCtrl : DINT;
		diStopperUnblkCtrlA : DINT;
		diStopperUnblkCtrlB : DINT;
		diMag1FixedClampCtrl : DINT;
		diMag1RemoteClampCtrl : DINT;
		diMag2FixedClampCtrl : DINT;
		diMag2RemoteClampCtrl : DINT;
		diMag3FixedClampCtrl : DINT;
		diMag3RemoteClampCtrl : DINT;
		diInShutterOpenCtrl : DINT;
		diInShutterCloseCtrl : DINT;
		diOutShutterOpenCtrl : DINT;
		diOutShutterCloseCtrl : DINT;
		diMag1ConvMtrIn : DINT;
		diMag1ConvMtrOut : DINT;
		diMag2ConvMtrIn : DINT;
		diMag2ConvMtrOut : DINT;
		diMag3ConvMtrIn : DINT;
		diMag3ConvMtrOut : DINT;
		diMag1SelClampCtrl : DINT;
		diMag2SelClampCtrl : DINT;
		diMag3SelClampCtrl : DINT;
		diPushConvMtrOn : DINT;
		diMag1WallEngageCtrl : DINT;
		diMag2WallEngageCtrl : DINT;
		diMag3WallEngageCtrl : DINT;
		diMag1SafetyBarRetCtrl : DINT;
		diMag2SafetyBarRetCtrl : DINT;
		diMag3SafetyBarRetCtrl : DINT;
		diSOT1MagError : DINT;
		diSOT1MagSizeLarge : DINT;
		diSOT1MagReady : DINT;
		diSOT1MagAvailable : DINT;
		diSOT2MagError : DINT;
		diSOT2MagSizeLarge : DINT;
		diSOT2MagReady : DINT;
		diSOT2MagAvailable : DINT;
		diSOT3MagError : DINT;
		diSOT3MagSizeLarge : DINT;
		diSOT3MagReady : DINT;
		diSOT3MagAvailable : DINT;
		diSOT4MagError : DINT;
		diSOT4MagSizeLarge : DINT;
		diSOT4MagReady : DINT;
		diSOT4MagAvailable : DINT;
		diMagAWOpenLimByp1 : DINT;
		diMagAWOpenLimByp2 : DINT;
		diMagAWOpenLimByp3 : DINT;
		diMagAWOpenLimByp4 : DINT;
		diMagAWSmallLimSen1 : DINT;
		diMagAWSmallLimSen2 : DINT;
		diMagAWSmallLimSen3 : DINT;
		diMagAWSmallLimSen4 : DINT;
		diMag1ReqToBring : DINT;
		diMag1ReqToGet : DINT;
		diMag2ReqToBring : DINT;
		diMag2ReqToGet : DINT;
		diMag3ReqToBring : DINT;
		diMag3ReqToGet : DINT;
		diMag4ReqToBring : DINT;
		diMag4ReqToGet : DINT;
		diMtrPshrExt : DINT;
		diMtrPshrRet : DINT;
		diMtrPshrOn : DINT;
		diMtrPshrBrakeRls : DINT;
		diMtrPshrSpdBinBit0 : DINT;
		diMtrPshrSpdBinBit1 : DINT;
		diMtrPshrSpdBinBit2 : DINT;
		diMtrPshrAlmRst : DINT;
		diInMagConvMtrOn : DINT;
		diOutMagConvMtrOn : DINT;
		diInMagConv2MtrOn : DINT;
		diOutMagConv2MtrOn : DINT;
		diEntTopStprUnblkCtrl : DINT; (*MagConv_Top*)
		diMidTopStprUnblkCtrl : DINT;
		diExtTopStprUnblkCtrl : DINT;
		diMidBtmStprUnblkCtrl : DINT;
		diExtBtmStprUnblkCtrl : DINT;
		diEntTopStprUnblkCtrl2 : DINT;
		diMidTopStprUnblkCtrl2 : DINT;
		diExtTopStprUnblkCtrl2 : DINT;
		diMidBtmStprUnblkCtrl2 : DINT;
		diExtBtmStprUnblkCtrl2 : DINT;
		diMtrPwrRly : DINT;
		diMag1FixedClampOpenCtrl : DINT;
		diMag1RemoteClampOpenCtrl : DINT;
		diMag2FixedClampOpenCtrl : DINT;
		diMag2RemoteClampOpenCtrl : DINT;
		diMag3FixedClampOpenCtrl : DINT;
		diMag3RemoteClampOpenCtrl : DINT;
		diOutShutterOpenCtrl2 : DINT;
		diOutShutterCloseCtrl2 : DINT;
		diOutShutterOpenCtrl3 : DINT;
		diOutShutterCloseCtrl3 : DINT;
		diBypCurtainSen : DINT;
		diRstCurtainSen : DINT;
		diBypCurtainPBLED : DINT;
		diInletStopperRetCtrl : DINT;
		diInletStopperExtCtrl : DINT;
		diScanTrigSig : DINT;
		diMag1ExitPCB : DINT;
		diMag2ExitPCB : DINT;
		diMag3ExitPCB : DINT;
		diMag1SelUnClampCtrl : DINT;
	END_STRUCT;
END_TYPE
```

### DOutput.var - Change By Project
```iecst
(*2019-01-08*)
(**)
(*Constant*)
VAR CONSTANT
	c_udiDOutputMax : UDINT := 200; (*Constant Digital Output Quantity (+1 For Damaged)(+1 For Spare)*)
END_VAR
(*Global*)
VAR
	g_tyDOutput : tyDigitalOutput;
END_VAR
```

### Program Logical/DOutput/DOutput (IEC, version 1.00.0) - 1.00.0 - (2018-12-01)

#### Cyclic.st - Change By Project
```iecst
(** 2019-03-29 **)
PROGRAM _CYCLIC
	Act_Background;

	IF bInitDone = FALSE THEN
		bInitDone	:= TRUE;

		Act_InitLocal;
		Act_InitGlobal;

	ELSIF bInitialDone = FALSE THEN
		bInitialDone	:= TRUE;

		Act_Initial;

	ELSE

		Act_LinkAction;
		Act_Action;
		Act_Link;
		Act_Main;
		Act_Background;

	END_IF

END_PROGRAM
```

#### Act_Background.st - Change By Project
```iecst
(** 2019-01-08 **)
ACTION Act_Background:

	//Resetting Physical Output
	memset(ADR(a_bPhysicalDO), 0, SIZEOF(a_bPhysicalDO));

	//Digital Output Mapping Physical Output With Config
	IF g_tyNtParamCurr.tyDOSettings.diSafetyRlyRst > 0 AND g_tyNtParamCurr.tyDOSettings.diSafetyRlyRst <= UDINT_TO_DINT(c_udiDOutputMax) THEN
		a_bPhysicalDO[g_tyNtParamCurr.tyDOSettings.diSafetyRlyRst]	:= g_tyRstErrOut.bSafetyRlyRst;
	END_IF

	IF g_tyNtParamCurr.tyDOSettings.diTLRed > 0 AND g_tyNtParamCurr.tyDOSettings.diTLRed <= UDINT_TO_DINT(c_udiDOutputMax) THEN
		a_bPhysicalDO[g_tyNtParamCurr.tyDOSettings.diTLRed]	:= g_tyTLBuz.bTLRed;
	END_IF

	IF g_tyNtParamCurr.tyDOSettings.diTLAmber > 0 AND g_tyNtParamCurr.tyDOSettings.diTLAmber <= UDINT_TO_DINT(c_udiDOutputMax) THEN
		a_bPhysicalDO[g_tyNtParamCurr.tyDOSettings.diTLAmber]	:= g_tyTLBuz.bTLAmber;
	END_IF

	IF g_tyNtParamCurr.tyDOSettings.diTLGreen > 0 AND g_tyNtParamCurr.tyDOSettings.diTLGreen <= UDINT_TO_DINT(c_udiDOutputMax) THEN
		a_bPhysicalDO[g_tyNtParamCurr.tyDOSettings.diTLGreen]	:= g_tyTLBuz.bTLGreen;
	END_IF

	IF g_tyNtParamCurr.tyDOSettings.diBuzzer > 0 AND g_tyNtParamCurr.tyDOSettings.diBuzzer <= UDINT_TO_DINT(c_udiDOutputMax) THEN
		a_bPhysicalDO[g_tyNtParamCurr.tyDOSettings.diBuzzer]	:= g_tyTLBuz.bBuzBeep;
	END_IF

	IF g_tyNtParamCurr.tyDOSettings.diUSBA > 0 AND g_tyNtParamCurr.tyDOSettings.diUSBA <= UDINT_TO_DINT(c_udiDOutputMax) THEN
		a_bPhysicalDO[g_tyNtParamCurr.tyDOSettings.diUSBA]	:= g_tyUSSMEMAA.bUSB;
	END_IF

	IF g_tyNtParamCurr.tyDOSettings.diUSBB > 0 AND g_tyNtParamCurr.tyDOSettings.diUSBB <= UDINT_TO_DINT(c_udiDOutputMax) THEN
		a_bPhysicalDO[g_tyNtParamCurr.tyDOSettings.diUSBB]	:= g_tyUSSMEMAB.bUSB;
	END_IF

	IF g_tyNtParamCurr.tyDOSettings.diOvenInfoSigA > 0 AND g_tyNtParamCurr.tyDOSettings.diOvenInfoSigA <= UDINT_TO_DINT(c_udiDOutputMax) THEN
		a_bPhysicalDO[g_tyNtParamCurr.tyDOSettings.diOvenInfoSigA]	:= g_tyOvenInfoA.bOvenAllow;
	END_IF

	IF g_tyNtParamCurr.tyDOSettings.diOvenInfoSigB > 0 AND g_tyNtParamCurr.tyDOSettings.diOvenInfoSigB <= UDINT_TO_DINT(c_udiDOutputMax) THEN
		a_bPhysicalDO[g_tyNtParamCurr.tyDOSettings.diOvenInfoSigB]	:= g_tyOvenInfoB.bOvenAllow;
	END_IF

	IF g_tyNtParamCurr.tyDOSettings.diPusherExtCtrl > 0 AND g_tyNtParamCurr.tyDOSettings.diPusherExtCtrl <= UDINT_TO_DINT(c_udiDOutputMax) THEN
		a_bPhysicalDO[g_tyNtParamCurr.tyDOSettings.diPusherExtCtrl]	:= g_tyPshrConv.bPshrExtCtrl;
	END_IF

	IF g_tyNtParamCurr.tyDOSettings.diStopperUnblkCtrlA > 0 AND g_tyNtParamCurr.tyDOSettings.diStopperUnblkCtrlA <= UDINT_TO_DINT(c_udiDOutputMax) THEN
		a_bPhysicalDO[g_tyNtParamCurr.tyDOSettings.diStopperUnblkCtrlA]	:= g_tyPneuStopperA.bRetCtrl;
	END_IF

	IF g_tyNtParamCurr.tyDOSettings.diStopperUnblkCtrlB > 0 AND g_tyNtParamCurr.tyDOSettings.diStopperUnblkCtrlB <= UDINT_TO_DINT(c_udiDOutputMax) THEN
		a_bPhysicalDO[g_tyNtParamCurr.tyDOSettings.diStopperUnblkCtrlB]	:= g_tyPneuStopperB.bRetCtrl;
	END_IF

	IF g_tyNtParamCurr.tyDOSettings.diMag1FixedClampCtrl > 0 AND g_tyNtParamCurr.tyDOSettings.diMag1FixedClampCtrl <= UDINT_TO_DINT(c_udiDOutputMax) THEN
		a_bPhysicalDO[g_tyNtParamCurr.tyDOSettings.diMag1FixedClampCtrl]	:= g_tyMagConv2Clp1.bFixClprClampCtrl;
	END_IF

	IF g_tyNtParamCurr.tyDOSettings.diMag1RemoteClampCtrl > 0 AND g_tyNtParamCurr.tyDOSettings.diMag1RemoteClampCtrl <= UDINT_TO_DINT(c_udiDOutputMax) THEN
		a_bPhysicalDO[g_tyNtParamCurr.tyDOSettings.diMag1RemoteClampCtrl]	:= g_tyMagConv2Clp1.bRemoteClampCtrl;
	END_IF

	IF g_tyNtParamCurr.tyDOSettings.diMag2FixedClampCtrl > 0 AND g_tyNtParamCurr.tyDOSettings.diMag2FixedClampCtrl <= UDINT_TO_DINT(c_udiDOutputMax) THEN
		a_bPhysicalDO[g_tyNtParamCurr.tyDOSettings.diMag2FixedClampCtrl]	:= g_tyMagConv2Clp2.bFixClprClampCtrl;
	END_IF

	IF g_tyNtParamCurr.tyDOSettings.diMag2RemoteClampCtrl > 0 AND g_tyNtParamCurr.tyDOSettings.diMag2RemoteClampCtrl <= UDINT_TO_DINT(c_udiDOutputMax) THEN
		a_bPhysicalDO[g_tyNtParamCurr.tyDOSettings.diMag2RemoteClampCtrl]	:= g_tyMagConv2Clp2.bRemoteClampCtrl;
	END_IF

	IF g_tyNtParamCurr.tyDOSettings.diMag3FixedClampCtrl > 0 AND g_tyNtParamCurr.tyDOSettings.diMag3FixedClampCtrl <= UDINT_TO_DINT(c_udiDOutputMax) THEN
		a_bPhysicalDO[g_tyNtParamCurr.tyDOSettings.diMag3FixedClampCtrl]	:= g_tyMagConv2Clp3.bFixClprClampCtrl;
	END_IF

	IF g_tyNtParamCurr.tyDOSettings.diMag3RemoteClampCtrl > 0 AND g_tyNtParamCurr.tyDOSettings.diMag3RemoteClampCtrl <= UDINT_TO_DINT(c_udiDOutputMax) THEN
		a_bPhysicalDO[g_tyNtParamCurr.tyDOSettings.diMag3RemoteClampCtrl]	:= g_tyMagConv2Clp3.bRemoteClampCtrl;
	END_IF

	IF bShutterTuning = FALSE THEN

			IF g_tyNtParamCurr.tyDOSettings.diInShutterOpenCtrl > 0 AND g_tyNtParamCurr.tyDOSettings.diInShutterOpenCtrl <= UDINT_TO_DINT(c_udiDOutputMax) THEN
				a_bPhysicalDO[g_tyNtParamCurr.tyDOSettings.diInShutterOpenCtrl]	:= p_bInShutterOpenCtrl;
			END_IF

			IF g_tyNtParamCurr.tyDOSettings.diInShutterCloseCtrl > 0 AND g_tyNtParamCurr.tyDOSettings.diInShutterCloseCtrl <= UDINT_TO_DINT(c_udiDOutputMax) THEN
				a_bPhysicalDO[g_tyNtParamCurr.tyDOSettings.diInShutterCloseCtrl]	:= p_bInShutterCloseCtrl;
			END_IF

			IF g_tyNtParamCurr.tyDOSettings.diOutShutterOpenCtrl > 0 AND g_tyNtParamCurr.tyDOSettings.diOutShutterOpenCtrl <= UDINT_TO_DINT(c_udiDOutputMax) THEN
				a_bPhysicalDO[g_tyNtParamCurr.tyDOSettings.diOutShutterOpenCtrl]	:= p_bOutShutterOpenCtrl;
			END_IF

			IF g_tyNtParamCurr.tyDOSettings.diOutShutterCloseCtrl > 0 AND g_tyNtParamCurr.tyDOSettings.diOutShutterCloseCtrl <= UDINT_TO_DINT(c_udiDOutputMax) THEN
				a_bPhysicalDO[g_tyNtParamCurr.tyDOSettings.diOutShutterCloseCtrl]	:= p_bOutShutterCloseCtrl;
			END_IF

			IF g_tyNtParamCurr.tyDOSettings.diOutShutterOpenCtrl2 > 0 AND g_tyNtParamCurr.tyDOSettings.diOutShutterOpenCtrl2 <= UDINT_TO_DINT(c_udiDOutputMax) THEN
				a_bPhysicalDO[g_tyNtParamCurr.tyDOSettings.diOutShutterOpenCtrl2]	:= p_bOutShutterOpenCtrl2;
			END_IF

			IF g_tyNtParamCurr.tyDOSettings.diOutShutterCloseCtrl2 > 0 AND g_tyNtParamCurr.tyDOSettings.diOutShutterCloseCtrl2 <= UDINT_TO_DINT(c_udiDOutputMax) THEN
				a_bPhysicalDO[g_tyNtParamCurr.tyDOSettings.diOutShutterCloseCtrl2]	:= p_bOutShutterCloseCtrl2;
			END_IF

			IF g_tyNtParamCurr.tyDOSettings.diOutShutterOpenCtrl3 > 0 AND g_tyNtParamCurr.tyDOSettings.diOutShutterOpenCtrl3 <= UDINT_TO_DINT(c_udiDOutputMax) THEN
				a_bPhysicalDO[g_tyNtParamCurr.tyDOSettings.diOutShutterOpenCtrl3]	:= p_bOutShutterOpenCtrl3;
			END_IF

			IF g_tyNtParamCurr.tyDOSettings.diOutShutterCloseCtrl3 > 0 AND g_tyNtParamCurr.tyDOSettings.diOutShutterCloseCtrl3 <= UDINT_TO_DINT(c_udiDOutputMax) THEN
				a_bPhysicalDO[g_tyNtParamCurr.tyDOSettings.diOutShutterCloseCtrl3]	:= p_bOutShutterCloseCtrl3;
			END_IF

	ELSE

		CASE usiShutterTuningStep OF
			0:
				a_bPhysicalDO[g_tyNtParamCurr.tyDOSettings.diInShutterOpenCtrl]	:= TRUE;
				a_bPhysicalDO[g_tyNtParamCurr.tyDOSettings.diOutShutterOpenCtrl]	:= TRUE;
				a_bPhysicalDO[g_tyNtParamCurr.tyDOSettings.diOutShutterOpenCtrl2]	:= TRUE;
				a_bPhysicalDO[g_tyNtParamCurr.tyDOSettings.diOutShutterOpenCtrl3]	:= TRUE;

				fbShutterTuneOpnTim(IN:= TRUE);
				IF fbShutterTuneOpnTim.Q THEN
					usiShutterTuningStep := 10;
					fbShutterTuneOpnTim(IN:= FALSE);
					a_bPhysicalDO[g_tyNtParamCurr.tyDOSettings.diInShutterOpenCtrl]	:= FALSE;
					a_bPhysicalDO[g_tyNtParamCurr.tyDOSettings.diOutShutterOpenCtrl]	:= FALSE;
					a_bPhysicalDO[g_tyNtParamCurr.tyDOSettings.diOutShutterOpenCtrl2]	:= FALSE;
					a_bPhysicalDO[g_tyNtParamCurr.tyDOSettings.diOutShutterOpenCtrl3]	:= FALSE;
				END_IF
			10:

				a_bPhysicalDO[g_tyNtParamCurr.tyDOSettings.diInShutterCloseCtrl]	:= TRUE;
				a_bPhysicalDO[g_tyNtParamCurr.tyDOSettings.diOutShutterCloseCtrl]	:= TRUE;
				a_bPhysicalDO[g_tyNtParamCurr.tyDOSettings.diOutShutterCloseCtrl2]:= TRUE;
				a_bPhysicalDO[g_tyNtParamCurr.tyDOSettings.diOutShutterCloseCtrl3]:= TRUE;

				fbShutterTuneClsTim(IN:= TRUE);
				IF fbShutterTuneClsTim.Q THEN
					usiShutterTuningStep := 0;
					fbShutterTuneClsTim(IN:= FALSE);
					a_bPhysicalDO[g_tyNtParamCurr.tyDOSettings.diInShutterCloseCtrl]	:= FALSE;
					a_bPhysicalDO[g_tyNtParamCurr.tyDOSettings.diOutShutterCloseCtrl]	:= FALSE;
					a_bPhysicalDO[g_tyNtParamCurr.tyDOSettings.diOutShutterCloseCtrl2]	:= FALSE;
					a_bPhysicalDO[g_tyNtParamCurr.tyDOSettings.diOutShutterCloseCtrl3]	:= FALSE;
				END_IF

		END_CASE
	END_IF

	IF g_tyNtParamCurr.tyDOSettings.diMag1ConvMtrIn > 0 AND g_tyNtParamCurr.tyDOSettings.diMag1ConvMtrIn <= UDINT_TO_DINT(c_udiDOutputMax) THEN
		a_bPhysicalDO[g_tyNtParamCurr.tyDOSettings.diMag1ConvMtrIn]	:= g_tyMagConv2Clp1.bMtrSigOnOrLToR;
	END_IF

	IF g_tyNtParamCurr.tyDOSettings.diMag1ConvMtrOut > 0 AND g_tyNtParamCurr.tyDOSettings.diMag1ConvMtrOut <= UDINT_TO_DINT(c_udiDOutputMax) THEN
		a_bPhysicalDO[g_tyNtParamCurr.tyDOSettings.diMag1ConvMtrOut]	:= g_tyMagConv2Clp1.bMtrDirOrRToL;
	END_IF

	IF g_tyNtParamCurr.tyDOSettings.diMag2ConvMtrIn > 0 AND g_tyNtParamCurr.tyDOSettings.diMag2ConvMtrIn <= UDINT_TO_DINT(c_udiDOutputMax) THEN
		a_bPhysicalDO[g_tyNtParamCurr.tyDOSettings.diMag2ConvMtrIn]	:= g_tyMagConv2Clp2.bMtrSigOnOrLToR;
	END_IF

	IF g_tyNtParamCurr.tyDOSettings.diMag2ConvMtrOut > 0 AND g_tyNtParamCurr.tyDOSettings.diMag2ConvMtrOut <= UDINT_TO_DINT(c_udiDOutputMax) THEN
		a_bPhysicalDO[g_tyNtParamCurr.tyDOSettings.diMag2ConvMtrOut]	:= g_tyMagConv2Clp2.bMtrDirOrRToL;
	END_IF

	IF g_tyNtParamCurr.tyDOSettings.diMag3ConvMtrIn > 0 AND g_tyNtParamCurr.tyDOSettings.diMag3ConvMtrIn <= UDINT_TO_DINT(c_udiDOutputMax) THEN
		a_bPhysicalDO[g_tyNtParamCurr.tyDOSettings.diMag3ConvMtrIn]	:= g_tyMagConv2Clp3.bMtrSigOnOrLToR;
	END_IF

	IF g_tyNtParamCurr.tyDOSettings.diMag3ConvMtrOut > 0 AND g_tyNtParamCurr.tyDOSettings.diMag3ConvMtrOut <= UDINT_TO_DINT(c_udiDOutputMax) THEN
		a_bPhysicalDO[g_tyNtParamCurr.tyDOSettings.diMag3ConvMtrOut]	:= g_tyMagConv2Clp3.bMtrDirOrRToL;
	END_IF

	IF g_tyNtParamCurr.tyDOSettings.diMag1SelClampCtrl > 0 AND g_tyNtParamCurr.tyDOSettings.diMag1SelClampCtrl <= UDINT_TO_DINT(c_udiDOutputMax) THEN
		a_bPhysicalDO[g_tyNtParamCurr.tyDOSettings.diMag1SelClampCtrl]	:= g_tyPneuSelClamp1.bRetCtrl;
	END_IF

	IF g_tyNtParamCurr.tyDOSettings.diMag2SelClampCtrl > 0 AND g_tyNtParamCurr.tyDOSettings.diMag2SelClampCtrl <= UDINT_TO_DINT(c_udiDOutputMax) THEN
		a_bPhysicalDO[g_tyNtParamCurr.tyDOSettings.diMag2SelClampCtrl]	:= g_tyPneuSelClamp2.bRetCtrl;
	END_IF

	IF g_tyNtParamCurr.tyDOSettings.diMag3SelClampCtrl > 0 AND g_tyNtParamCurr.tyDOSettings.diMag3SelClampCtrl <= UDINT_TO_DINT(c_udiDOutputMax) THEN
		a_bPhysicalDO[g_tyNtParamCurr.tyDOSettings.diMag3SelClampCtrl]	:= g_tyPneuSelClamp3.bRetCtrl;
	END_IF

	IF g_tyNtParamCurr.tyDOSettings.diMag1SelUnClampCtrl > 0 AND g_tyNtParamCurr.tyDOSettings.diMag1SelUnClampCtrl <= UDINT_TO_DINT(c_udiDOutputMax) THEN
		a_bPhysicalDO[g_tyNtParamCurr.tyDOSettings.diMag1SelUnClampCtrl]	:= g_tyPneuSelClamp1.bExtCtrl;
	END_IF

//	IF g_tyNtParamCurr.tyDOSettings.diMag2SelUnClampCtrl > 0 AND g_tyNtParamCurr.tyDOSettings.diMag2SelUnClampCtrl <= UDINT_TO_DINT(c_udiDOutputMax) THEN
//		a_bPhysicalDO[g_tyNtParamCurr.tyDOSettings.diMag2SelUnClampCtrl]	:= g_tyPneuSelClamp2.bExtCtrl;
//	END_IF
//
//	IF g_tyNtParamCurr.tyDOSettings.diMag3SelUnClampCtrl > 0 AND g_tyNtParamCurr.tyDOSettings.diMag3SelUnClampCtrl <= UDINT_TO_DINT(c_udiDOutputMax) THEN
//		a_bPhysicalDO[g_tyNtParamCurr.tyDOSettings.diMag3SelUnClampCtrl]	:= g_tyPneuSelClamp3.bExtCtrl;
//	END_IF

	IF g_tyNtParamCurr.tyDOSettings.diPushConvMtrOn > 0 AND g_tyNtParamCurr.tyDOSettings.diPushConvMtrOn <= UDINT_TO_DINT(c_udiDOutputMax) THEN
		a_bPhysicalDO[g_tyNtParamCurr.tyDOSettings.diPushConvMtrOn]	:= g_tyPshrConv.bMtrSigOnOrLToR;
	END_IF

	IF g_tyNtParamCurr.tyDOSettings.diMag1SafetyBarRetCtrl > 0 AND g_tyNtParamCurr.tyDOSettings.diMag1SafetyBarRetCtrl <= UDINT_TO_DINT(c_udiDOutputMax) THEN
		a_bPhysicalDO[g_tyNtParamCurr.tyDOSettings.diMag1SafetyBarRetCtrl]	:= g_tyPneuMag1SafetyBar.bRetCtrl;
	END_IF

	IF g_tyNtParamCurr.tyDOSettings.diMag2SafetyBarRetCtrl > 0 AND g_tyNtParamCurr.tyDOSettings.diMag2SafetyBarRetCtrl <= UDINT_TO_DINT(c_udiDOutputMax) THEN
		a_bPhysicalDO[g_tyNtParamCurr.tyDOSettings.diMag2SafetyBarRetCtrl]	:= g_tyPneuMag2SafetyBar.bRetCtrl;
	END_IF

	IF g_tyNtParamCurr.tyDOSettings.diMag3SafetyBarRetCtrl > 0 AND g_tyNtParamCurr.tyDOSettings.diMag3SafetyBarRetCtrl <= UDINT_TO_DINT(c_udiDOutputMax) THEN
		a_bPhysicalDO[g_tyNtParamCurr.tyDOSettings.diMag3SafetyBarRetCtrl]	:= g_tyPneuMag3SafetyBar.bRetCtrl;
	END_IF

	IF g_tyNtParamCurr.tyDOSettings.diMag1WallEngageCtrl > 0 AND g_tyNtParamCurr.tyDOSettings.diMag1WallEngageCtrl <= UDINT_TO_DINT(c_udiDOutputMax) THEN
		a_bPhysicalDO[g_tyNtParamCurr.tyDOSettings.diMag1WallEngageCtrl]	:= g_tyPneuMag1AWEngage.bExtCtrl;
	END_IF

	IF g_tyNtParamCurr.tyDOSettings.diMag2WallEngageCtrl > 0 AND g_tyNtParamCurr.tyDOSettings.diMag2WallEngageCtrl <= UDINT_TO_DINT(c_udiDOutputMax) THEN
		a_bPhysicalDO[g_tyNtParamCurr.tyDOSettings.diMag2WallEngageCtrl]	:= g_tyPneuMag2AWEngage.bExtCtrl;
	END_IF

	IF g_tyNtParamCurr.tyDOSettings.diMag3WallEngageCtrl > 0 AND g_tyNtParamCurr.tyDOSettings.diMag3WallEngageCtrl <= UDINT_TO_DINT(c_udiDOutputMax) THEN
		a_bPhysicalDO[g_tyNtParamCurr.tyDOSettings.diMag3WallEngageCtrl]	:= g_tyPneuMag3AWEngage.bExtCtrl;
	END_IF

	IF bAgvComIODisabled = FALSE THEN
			//SOT Configuration
			IF g_tyNtParamCurr.tyDOSettings.diSOT1MagError > 0 AND g_tyNtParamCurr.tyDOSettings.diSOT1MagError <= UDINT_TO_DINT(c_udiDOutputMax) THEN
				a_bPhysicalDO[g_tyNtParamCurr.tyDOSettings.diSOT1MagError]				:= p_bSOTMagError1;
			END_IF

			IF g_tyNtParamCurr.tyDOSettings.diSOT1MagSizeLarge > 0 AND g_tyNtParamCurr.tyDOSettings.diSOT1MagSizeLarge <= UDINT_TO_DINT(c_udiDOutputMax) THEN
				a_bPhysicalDO[g_tyNtParamCurr.tyDOSettings.diSOT1MagSizeLarge]				:= p_bSOTMagSizeLarge1;
			END_IF

			IF g_tyNtParamCurr.tyDOSettings.diSOT1MagReady > 0 AND g_tyNtParamCurr.tyDOSettings.diSOT1MagReady <= UDINT_TO_DINT(c_udiDOutputMax) THEN
				a_bPhysicalDO[g_tyNtParamCurr.tyDOSettings.diSOT1MagReady]				:= p_bSOTMagReady1;
			END_IF

			IF g_tyNtParamCurr.tyDOSettings.diSOT1MagAvailable > 0 AND g_tyNtParamCurr.tyDOSettings.diSOT1MagAvailable <= UDINT_TO_DINT(c_udiDOutputMax) THEN
				a_bPhysicalDO[g_tyNtParamCurr.tyDOSettings.diSOT1MagAvailable]				:= p_bSOTMagAvailable1;
			END_IF

			IF g_tyNtParamCurr.tyDOSettings.diSOT2MagError > 0 AND g_tyNtParamCurr.tyDOSettings.diSOT2MagError <= UDINT_TO_DINT(c_udiDOutputMax) THEN
				a_bPhysicalDO[g_tyNtParamCurr.tyDOSettings.diSOT2MagError]				:= p_bSOTMagError2;
			END_IF

			IF g_tyNtParamCurr.tyDOSettings.diSOT2MagSizeLarge > 0 AND g_tyNtParamCurr.tyDOSettings.diSOT2MagSizeLarge <= UDINT_TO_DINT(c_udiDOutputMax) THEN
				a_bPhysicalDO[g_tyNtParamCurr.tyDOSettings.diSOT2MagSizeLarge]				:= p_bSOTMagSizeLarge2;
			END_IF

			IF g_tyNtParamCurr.tyDOSettings.diSOT2MagReady > 0 AND g_tyNtParamCurr.tyDOSettings.diSOT2MagReady <= UDINT_TO_DINT(c_udiDOutputMax) THEN
				a_bPhysicalDO[g_tyNtParamCurr.tyDOSettings.diSOT2MagReady]				:= p_bSOTMagReady2;
			END_IF

			IF g_tyNtParamCurr.tyDOSettings.diSOT2MagAvailable > 0 AND g_tyNtParamCurr.tyDOSettings.diSOT2MagAvailable <= UDINT_TO_DINT(c_udiDOutputMax) THEN
				a_bPhysicalDO[g_tyNtParamCurr.tyDOSettings.diSOT2MagAvailable]				:= p_bSOTMagAvailable2;
			END_IF

			IF g_tyNtParamCurr.tyDOSettings.diSOT3MagError > 0 AND g_tyNtParamCurr.tyDOSettings.diSOT3MagError <= UDINT_TO_DINT(c_udiDOutputMax) THEN
				a_bPhysicalDO[g_tyNtParamCurr.tyDOSettings.diSOT3MagError]				:= p_bSOTMagError3;
			END_IF

			IF g_tyNtParamCurr.tyDOSettings.diSOT3MagSizeLarge > 0 AND g_tyNtParamCurr.tyDOSettings.diSOT3MagSizeLarge <= UDINT_TO_DINT(c_udiDOutputMax) THEN
				a_bPhysicalDO[g_tyNtParamCurr.tyDOSettings.diSOT3MagSizeLarge]				:= p_bSOTMagSizeLarge3;
			END_IF

			IF g_tyNtParamCurr.tyDOSettings.diSOT3MagReady > 0 AND g_tyNtParamCurr.tyDOSettings.diSOT3MagReady <= UDINT_TO_DINT(c_udiDOutputMax) THEN
				a_bPhysicalDO[g_tyNtParamCurr.tyDOSettings.diSOT3MagReady]				:= p_bSOTMagReady3;
			END_IF

			IF g_tyNtParamCurr.tyDOSettings.diSOT3MagAvailable > 0 AND g_tyNtParamCurr.tyDOSettings.diSOT3MagAvailable <= UDINT_TO_DINT(c_udiDOutputMax) THEN
				a_bPhysicalDO[g_tyNtParamCurr.tyDOSettings.diSOT3MagAvailable]				:= p_bSOTMagAvailable3;
			END_IF

			IF g_tyNtParamCurr.tyDOSettings.diSOT4MagError > 0 AND g_tyNtParamCurr.tyDOSettings.diSOT4MagError <= UDINT_TO_DINT(c_udiDOutputMax) THEN
				a_bPhysicalDO[g_tyNtParamCurr.tyDOSettings.diSOT4MagError]				:= p_bSOTMagError4;
			END_IF

			IF g_tyNtParamCurr.tyDOSettings.diSOT4MagSizeLarge > 0 AND g_tyNtParamCurr.tyDOSettings.diSOT4MagSizeLarge <= UDINT_TO_DINT(c_udiDOutputMax) THEN
				a_bPhysicalDO[g_tyNtParamCurr.tyDOSettings.diSOT4MagSizeLarge]				:= p_bSOTMagSizeLarge4;
			END_IF

			IF g_tyNtParamCurr.tyDOSettings.diSOT4MagReady > 0 AND g_tyNtParamCurr.tyDOSettings.diSOT4MagReady <= UDINT_TO_DINT(c_udiDOutputMax) THEN
				a_bPhysicalDO[g_tyNtParamCurr.tyDOSettings.diSOT4MagReady]				:= p_bSOTMagReady4;
			END_IF

			IF g_tyNtParamCurr.tyDOSettings.diSOT4MagAvailable > 0 AND g_tyNtParamCurr.tyDOSettings.diSOT4MagAvailable <= UDINT_TO_DINT(c_udiDOutputMax) THEN
				a_bPhysicalDO[g_tyNtParamCurr.tyDOSettings.diSOT4MagAvailable]				:= p_bSOTMagAvailable4;
			END_IF
	ELSE
			a_bPhysicalDO[g_tyNtParamCurr.tyDOSettings.diSOT1MagError] := FALSE;
			a_bPhysicalDO[g_tyNtParamCurr.tyDOSettings.diSOT2MagError] := FALSE;
			a_bPhysicalDO[g_tyNtParamCurr.tyDOSettings.diSOT3MagError] := FALSE;
			a_bPhysicalDO[g_tyNtParamCurr.tyDOSettings.diSOT4MagError] := FALSE;
			a_bPhysicalDO[g_tyNtParamCurr.tyDOSettings.diSOT1MagSizeLarge] := FALSE;
			a_bPhysicalDO[g_tyNtParamCurr.tyDOSettings.diSOT2MagSizeLarge] := FALSE;
			a_bPhysicalDO[g_tyNtParamCurr.tyDOSettings.diSOT3MagSizeLarge] := FALSE;
			a_bPhysicalDO[g_tyNtParamCurr.tyDOSettings.diSOT4MagSizeLarge] := FALSE;
			a_bPhysicalDO[g_tyNtParamCurr.tyDOSettings.diSOT1MagReady] := FALSE;
			a_bPhysicalDO[g_tyNtParamCurr.tyDOSettings.diSOT2MagReady] := FALSE;
			a_bPhysicalDO[g_tyNtParamCurr.tyDOSettings.diSOT3MagReady] := FALSE;
			a_bPhysicalDO[g_tyNtParamCurr.tyDOSettings.diSOT4MagReady] := FALSE;
			a_bPhysicalDO[g_tyNtParamCurr.tyDOSettings.diSOT1MagAvailable] := FALSE;
			a_bPhysicalDO[g_tyNtParamCurr.tyDOSettings.diSOT2MagAvailable] := FALSE;
			a_bPhysicalDO[g_tyNtParamCurr.tyDOSettings.diSOT3MagAvailable] := FALSE;
			a_bPhysicalDO[g_tyNtParamCurr.tyDOSettings.diSOT4MagAvailable] := FALSE;
	END_IF

	IF g_tyNtParamCurr.tyDOSettings.diMagAWOpenLimByp1 > 0 AND g_tyNtParamCurr.tyDOSettings.diMagAWOpenLimByp1 <= UDINT_TO_DINT(c_udiDOutputMax) THEN
		a_bPhysicalDO[g_tyNtParamCurr.tyDOSettings.diMagAWOpenLimByp1]				:= bMagAWOpenLimByp1;
	END_IF

	IF g_tyNtParamCurr.tyDOSettings.diMagAWOpenLimByp2 > 0 AND g_tyNtParamCurr.tyDOSettings.diMagAWOpenLimByp2 <= UDINT_TO_DINT(c_udiDOutputMax) THEN
		a_bPhysicalDO[g_tyNtParamCurr.tyDOSettings.diMagAWOpenLimByp2]				:= bMagAWOpenLimByp2;
	END_IF

	IF g_tyNtParamCurr.tyDOSettings.diMagAWOpenLimByp3 > 0 AND g_tyNtParamCurr.tyDOSettings.diMagAWOpenLimByp3 <= UDINT_TO_DINT(c_udiDOutputMax) THEN
		a_bPhysicalDO[g_tyNtParamCurr.tyDOSettings.diMagAWOpenLimByp3]				:= bMagAWOpenLimByp3;
	END_IF

	IF g_tyNtParamCurr.tyDOSettings.diMagAWOpenLimByp4 > 0 AND g_tyNtParamCurr.tyDOSettings.diMagAWOpenLimByp4 <= UDINT_TO_DINT(c_udiDOutputMax) THEN
		a_bPhysicalDO[g_tyNtParamCurr.tyDOSettings.diMagAWOpenLimByp4]				:= bMagAWOpenLimByp4;
	END_IF

	IF g_tyNtParamCurr.tyDOSettings.diMagAWSmallLimSen1 > 0 AND g_tyNtParamCurr.tyDOSettings.diMagAWSmallLimSen1 <= UDINT_TO_DINT(c_udiDOutputMax) THEN
		a_bPhysicalDO[g_tyNtParamCurr.tyDOSettings.diMagAWSmallLimSen1]				:= bMagAWSmallLimSen1;
	END_IF

	IF g_tyNtParamCurr.tyDOSettings.diMagAWSmallLimSen2 > 0 AND g_tyNtParamCurr.tyDOSettings.diMagAWSmallLimSen2 <= UDINT_TO_DINT(c_udiDOutputMax) THEN
		a_bPhysicalDO[g_tyNtParamCurr.tyDOSettings.diMagAWSmallLimSen2]				:= bMagAWSmallLimSen2;
	END_IF

	IF g_tyNtParamCurr.tyDOSettings.diMagAWSmallLimSen3 > 0 AND g_tyNtParamCurr.tyDOSettings.diMagAWSmallLimSen3 <= UDINT_TO_DINT(c_udiDOutputMax) THEN
		a_bPhysicalDO[g_tyNtParamCurr.tyDOSettings.diMagAWSmallLimSen3]				:= bMagAWSmallLimSen3;
	END_IF

	IF g_tyNtParamCurr.tyDOSettings.diMagAWSmallLimSen4 > 0 AND g_tyNtParamCurr.tyDOSettings.diMagAWSmallLimSen4 <= UDINT_TO_DINT(c_udiDOutputMax) THEN
		a_bPhysicalDO[g_tyNtParamCurr.tyDOSettings.diMagAWSmallLimSen4]				:= bMagAWSmallLimSen4;
	END_IF

	IF p_eLinkAGVComProtocol = McSetAGVCommHardIO THEN
		//AIV signals Get/Bring Magazine
		IF g_tyNtParamCurr.tyDOSettings.diMag1ReqToBring > 0 AND g_tyNtParamCurr.tyDOSettings.diMag1ReqToBring <= UDINT_TO_DINT(c_udiDOutputMax) THEN
			a_bPhysicalDO[g_tyNtParamCurr.tyDOSettings.diMag1ReqToBring]				:= bRequestToBring1;
		END_IF

		IF g_tyNtParamCurr.tyDOSettings.diMag1ReqToGet > 0 AND g_tyNtParamCurr.tyDOSettings.diMag1ReqToGet <= UDINT_TO_DINT(c_udiDOutputMax) THEN
			a_bPhysicalDO[g_tyNtParamCurr.tyDOSettings.diMag1ReqToGet]				:= bRequestToGet1;
		END_IF

		IF g_tyNtParamCurr.tyDOSettings.diMag2ReqToBring > 0 AND g_tyNtParamCurr.tyDOSettings.diMag2ReqToBring <= UDINT_TO_DINT(c_udiDOutputMax) THEN
			a_bPhysicalDO[g_tyNtParamCurr.tyDOSettings.diMag2ReqToBring]				:= bRequestToBring2;
		END_IF

		IF g_tyNtParamCurr.tyDOSettings.diMag2ReqToGet > 0 AND g_tyNtParamCurr.tyDOSettings.diMag2ReqToGet <= UDINT_TO_DINT(c_udiDOutputMax) THEN
			a_bPhysicalDO[g_tyNtParamCurr.tyDOSettings.diMag2ReqToGet]				:= bRequestToGet2;
		END_IF

		IF g_tyNtParamCurr.tyDOSettings.diMag3ReqToBring > 0 AND g_tyNtParamCurr.tyDOSettings.diMag3ReqToBring <= UDINT_TO_DINT(c_udiDOutputMax) THEN
			a_bPhysicalDO[g_tyNtParamCurr.tyDOSettings.diMag3ReqToBring]				:= bRequestToBring3;
		END_IF

		IF g_tyNtParamCurr.tyDOSettings.diMag3ReqToGet > 0 AND g_tyNtParamCurr.tyDOSettings.diMag3ReqToGet <= UDINT_TO_DINT(c_udiDOutputMax) THEN
			a_bPhysicalDO[g_tyNtParamCurr.tyDOSettings.diMag3ReqToGet]				:= bRequestToGet3;
		END_IF

		IF g_tyNtParamCurr.tyDOSettings.diMag4ReqToBring > 0 AND g_tyNtParamCurr.tyDOSettings.diMag4ReqToBring <= UDINT_TO_DINT(c_udiDOutputMax) THEN
			a_bPhysicalDO[g_tyNtParamCurr.tyDOSettings.diMag4ReqToBring]				:= bRequestToBring4;
		END_IF

		IF g_tyNtParamCurr.tyDOSettings.diMag4ReqToGet > 0 AND g_tyNtParamCurr.tyDOSettings.diMag4ReqToGet <= UDINT_TO_DINT(c_udiDOutputMax) THEN
			a_bPhysicalDO[g_tyNtParamCurr.tyDOSettings.diMag4ReqToGet]				:= bRequestToGet4;
		END_IF
	ELSE
		a_bPhysicalDO[g_tyNtParamCurr.tyDOSettings.diMag1ReqToBring] := FALSE;
		a_bPhysicalDO[g_tyNtParamCurr.tyDOSettings.diMag1ReqToGet] := FALSE;
		a_bPhysicalDO[g_tyNtParamCurr.tyDOSettings.diMag2ReqToBring] := FALSE;
		a_bPhysicalDO[g_tyNtParamCurr.tyDOSettings.diMag2ReqToGet] := FALSE;
		a_bPhysicalDO[g_tyNtParamCurr.tyDOSettings.diMag3ReqToBring] := FALSE;
		a_bPhysicalDO[g_tyNtParamCurr.tyDOSettings.diMag3ReqToGet] := FALSE;
		a_bPhysicalDO[g_tyNtParamCurr.tyDOSettings.diMag4ReqToBring] := FALSE;
		a_bPhysicalDO[g_tyNtParamCurr.tyDOSettings.diMag4ReqToGet] := FALSE;
	END_IF

	IF g_tyNtParamCurr.tyDOSettings.diMtrPshrExt > 0 AND g_tyNtParamCurr.tyDOSettings.diMtrPshrExt <= UDINT_TO_DINT(c_udiDOutputMax) THEN
		a_bPhysicalDO[g_tyNtParamCurr.tyDOSettings.diMtrPshrExt]	:= p_bMtrPshrExt;
	END_IF

	IF g_tyNtParamCurr.tyDOSettings.diMtrPshrRet > 0 AND g_tyNtParamCurr.tyDOSettings.diMtrPshrRet <= UDINT_TO_DINT(c_udiDOutputMax) THEN
		a_bPhysicalDO[g_tyNtParamCurr.tyDOSettings.diMtrPshrRet]	:= p_bMtrPshrRet;
	END_IF

	IF g_tyNtParamCurr.tyDOSettings.diMtrPshrOn > 0 AND g_tyNtParamCurr.tyDOSettings.diMtrPshrOn <= UDINT_TO_DINT(c_udiDOutputMax) THEN
		a_bPhysicalDO[g_tyNtParamCurr.tyDOSettings.diMtrPshrOn]	:= p_bMtrPshrOn;
	END_IF

	IF g_tyNtParamCurr.tyDOSettings.diMtrPshrBrakeRls > 0 AND g_tyNtParamCurr.tyDOSettings.diMtrPshrBrakeRls <= UDINT_TO_DINT(c_udiDOutputMax) THEN
		a_bPhysicalDO[g_tyNtParamCurr.tyDOSettings.diMtrPshrBrakeRls]	:= p_bMtrPshrBrakeRls;
	END_IF

	IF g_tyNtParamCurr.tyDOSettings.diMtrPshrSpdBinBit0 > 0 AND g_tyNtParamCurr.tyDOSettings.diMtrPshrSpdBinBit0 <= UDINT_TO_DINT(c_udiDOutputMax) THEN
		a_bPhysicalDO[g_tyNtParamCurr.tyDOSettings.diMtrPshrSpdBinBit0]	:= p_bMtrPshrSpdBinBit0;
	END_IF

	IF g_tyNtParamCurr.tyDOSettings.diMtrPshrSpdBinBit1 > 0 AND g_tyNtParamCurr.tyDOSettings.diMtrPshrSpdBinBit1 <= UDINT_TO_DINT(c_udiDOutputMax) THEN
		a_bPhysicalDO[g_tyNtParamCurr.tyDOSettings.diMtrPshrSpdBinBit1]	:= p_bMtrPshrSpdBinBit1;
	END_IF

	IF g_tyNtParamCurr.tyDOSettings.diMtrPshrSpdBinBit2 > 0 AND g_tyNtParamCurr.tyDOSettings.diMtrPshrSpdBinBit2 <= UDINT_TO_DINT(c_udiDOutputMax) THEN
		a_bPhysicalDO[g_tyNtParamCurr.tyDOSettings.diMtrPshrSpdBinBit2]	:= p_bMtrPshrSpdBinBit2;
	END_IF

	IF g_tyNtParamCurr.tyDOSettings.diMtrPshrAlmRst > 0 AND g_tyNtParamCurr.tyDOSettings.diMtrPshrAlmRst <= UDINT_TO_DINT(c_udiDOutputMax) THEN
		a_bPhysicalDO[g_tyNtParamCurr.tyDOSettings.diMtrPshrAlmRst]	:= p_bMtrPshrAlmRst;
	END_IF

	IF g_tyNtParamCurr.tyDOSettings.diInMagConvMtrOn > 0 AND g_tyNtParamCurr.tyDOSettings.diInMagConvMtrOn <= UDINT_TO_DINT(c_udiDOutputMax) THEN
		a_bPhysicalDO[g_tyNtParamCurr.tyDOSettings.diInMagConvMtrOn]	:= p_bInMagConvMtrOn;
	END_IF

	IF g_tyNtParamCurr.tyDOSettings.diOutMagConvMtrOn > 0 AND g_tyNtParamCurr.tyDOSettings.diOutMagConvMtrOn <= UDINT_TO_DINT(c_udiDOutputMax) THEN
		a_bPhysicalDO[g_tyNtParamCurr.tyDOSettings.diOutMagConvMtrOn]	:= p_bOutMagConvMtrOn;
	END_IF

	IF g_tyNtParamCurr.tyDOSettings.diInMagConv2MtrOn > 0 AND g_tyNtParamCurr.tyDOSettings.diInMagConv2MtrOn <= UDINT_TO_DINT(c_udiDOutputMax) THEN
		a_bPhysicalDO[g_tyNtParamCurr.tyDOSettings.diInMagConv2MtrOn]	:= p_bInMagConv2MtrOn;
	END_IF

	IF g_tyNtParamCurr.tyDOSettings.diOutMagConv2MtrOn > 0 AND g_tyNtParamCurr.tyDOSettings.diOutMagConv2MtrOn <= UDINT_TO_DINT(c_udiDOutputMax) THEN
		a_bPhysicalDO[g_tyNtParamCurr.tyDOSettings.diOutMagConv2MtrOn]	:= p_bOutMagConv2MtrOn;
	END_IF

	IF g_tyNtParamCurr.tyDOSettings.diEntTopStprUnblkCtrl > 0 AND g_tyNtParamCurr.tyDOSettings.diEntTopStprUnblkCtrl <= UDINT_TO_DINT(c_udiDOutputMax) THEN
		a_bPhysicalDO[g_tyNtParamCurr.tyDOSettings.diEntTopStprUnblkCtrl]	:= p_bEntTopStprUnblkCtrl;
	END_IF
	IF g_tyNtParamCurr.tyDOSettings.diMidTopStprUnblkCtrl > 0 AND g_tyNtParamCurr.tyDOSettings.diMidTopStprUnblkCtrl <= UDINT_TO_DINT(c_udiDOutputMax) THEN
		a_bPhysicalDO[g_tyNtParamCurr.tyDOSettings.diMidTopStprUnblkCtrl]	:= p_bMidTopStprUnblkCtrl;
	END_IF
	IF g_tyNtParamCurr.tyDOSettings.diExtTopStprUnblkCtrl > 0 AND g_tyNtParamCurr.tyDOSettings.diExtTopStprUnblkCtrl <= UDINT_TO_DINT(c_udiDOutputMax) THEN
		a_bPhysicalDO[g_tyNtParamCurr.tyDOSettings.diExtTopStprUnblkCtrl]	:= p_bExtTopStprUnblkCtrl;
	END_IF
	IF g_tyNtParamCurr.tyDOSettings.diMidBtmStprUnblkCtrl > 0 AND g_tyNtParamCurr.tyDOSettings.diMidBtmStprUnblkCtrl <= UDINT_TO_DINT(c_udiDOutputMax) THEN
		a_bPhysicalDO[g_tyNtParamCurr.tyDOSettings.diMidBtmStprUnblkCtrl]	:= p_bMidBtmStprUnblkCtrl;
	END_IF
	IF g_tyNtParamCurr.tyDOSettings.diExtBtmStprUnblkCtrl > 0 AND g_tyNtParamCurr.tyDOSettings.diExtBtmStprUnblkCtrl <= UDINT_TO_DINT(c_udiDOutputMax) THEN
		a_bPhysicalDO[g_tyNtParamCurr.tyDOSettings.diExtBtmStprUnblkCtrl]	:= p_bExtBtmStprUnblkCtrl;
	END_IF

	IF g_tyNtParamCurr.tyDOSettings.diEntTopStprUnblkCtrl2 > 0 AND g_tyNtParamCurr.tyDOSettings.diEntTopStprUnblkCtrl2 <= UDINT_TO_DINT(c_udiDOutputMax) THEN
		a_bPhysicalDO[g_tyNtParamCurr.tyDOSettings.diEntTopStprUnblkCtrl2]	:= p_bEntTopStprUnblkCtrl2;
	END_IF
	IF g_tyNtParamCurr.tyDOSettings.diMidTopStprUnblkCtrl2 > 0 AND g_tyNtParamCurr.tyDOSettings.diMidTopStprUnblkCtrl2 <= UDINT_TO_DINT(c_udiDOutputMax) THEN
		a_bPhysicalDO[g_tyNtParamCurr.tyDOSettings.diMidTopStprUnblkCtrl2]	:= p_bMidTopStprUnblkCtrl2;
	END_IF
	IF g_tyNtParamCurr.tyDOSettings.diExtTopStprUnblkCtrl2 > 0 AND g_tyNtParamCurr.tyDOSettings.diExtTopStprUnblkCtrl2 <= UDINT_TO_DINT(c_udiDOutputMax) THEN
		a_bPhysicalDO[g_tyNtParamCurr.tyDOSettings.diExtTopStprUnblkCtrl2]	:= p_bExtTopStprUnblkCtrl2;
	END_IF
	IF g_tyNtParamCurr.tyDOSettings.diMidBtmStprUnblkCtrl2 > 0 AND g_tyNtParamCurr.tyDOSettings.diMidBtmStprUnblkCtrl2 <= UDINT_TO_DINT(c_udiDOutputMax) THEN
		a_bPhysicalDO[g_tyNtParamCurr.tyDOSettings.diMidBtmStprUnblkCtrl2]	:= p_bMidBtmStprUnblkCtrl2;
	END_IF
	IF g_tyNtParamCurr.tyDOSettings.diExtBtmStprUnblkCtrl2 > 0 AND g_tyNtParamCurr.tyDOSettings.diExtBtmStprUnblkCtrl2 <= UDINT_TO_DINT(c_udiDOutputMax) THEN
		a_bPhysicalDO[g_tyNtParamCurr.tyDOSettings.diExtBtmStprUnblkCtrl2]	:= p_bExtBtmStprUnblkCtrl2;
	END_IF

	IF g_tyNtParamCurr.tyDOSettings.diExtBtmStprUnblkCtrl2 > 0 AND g_tyNtParamCurr.tyDOSettings.diExtBtmStprUnblkCtrl2 <= UDINT_TO_DINT(c_udiDOutputMax) THEN
		a_bPhysicalDO[g_tyNtParamCurr.tyDOSettings.diExtBtmStprUnblkCtrl2]	:= p_bExtBtmStprUnblkCtrl2;
	END_IF

	IF g_tyNtParamCurr.tyDOSettings.diMtrPwrRly > 0 AND g_tyNtParamCurr.tyDOSettings.diMtrPwrRly <= UDINT_TO_DINT(c_udiDOutputMax) THEN
		a_bPhysicalDO[g_tyNtParamCurr.tyDOSettings.diMtrPwrRly]						:= p_bMtrPwrRly;
	END_IF

	IF g_tyNtParamCurr.tyDOSettings.diMag1FixedClampOpenCtrl > 0 AND g_tyNtParamCurr.tyDOSettings.diMag1FixedClampOpenCtrl <= UDINT_TO_DINT(c_udiDOutputMax) THEN
		a_bPhysicalDO[g_tyNtParamCurr.tyDOSettings.diMag1FixedClampOpenCtrl]	:= NOT p_bMag1FixedClampOpenCtrl;
	END_IF

	IF g_tyNtParamCurr.tyDOSettings.diMag1RemoteClampOpenCtrl > 0 AND g_tyNtParamCurr.tyDOSettings.diMag1RemoteClampOpenCtrl <= UDINT_TO_DINT(c_udiDOutputMax) THEN
		a_bPhysicalDO[g_tyNtParamCurr.tyDOSettings.diMag1RemoteClampOpenCtrl]	:= NOT p_bMag1RemoteClampOpenCtrl;
	END_IF

	IF g_tyNtParamCurr.tyDOSettings.diMag2FixedClampOpenCtrl > 0 AND g_tyNtParamCurr.tyDOSettings.diMag2FixedClampOpenCtrl <= UDINT_TO_DINT(c_udiDOutputMax) THEN
		a_bPhysicalDO[g_tyNtParamCurr.tyDOSettings.diMag2FixedClampOpenCtrl]	:= NOT p_bMag2FixedClampOpenCtrl;
	END_IF

	IF g_tyNtParamCurr.tyDOSettings.diMag2RemoteClampOpenCtrl > 0 AND g_tyNtParamCurr.tyDOSettings.diMag2RemoteClampOpenCtrl <= UDINT_TO_DINT(c_udiDOutputMax) THEN
		a_bPhysicalDO[g_tyNtParamCurr.tyDOSettings.diMag2RemoteClampOpenCtrl]	:= NOT p_bMag2RemoteClampOpenCtrl;
	END_IF

	IF g_tyNtParamCurr.tyDOSettings.diMag3FixedClampOpenCtrl > 0 AND g_tyNtParamCurr.tyDOSettings.diMag3FixedClampOpenCtrl <= UDINT_TO_DINT(c_udiDOutputMax) THEN
		a_bPhysicalDO[g_tyNtParamCurr.tyDOSettings.diMag3FixedClampOpenCtrl]	:= NOT p_bMag3FixedClampOpenCtrl;
	END_IF

	IF g_tyNtParamCurr.tyDOSettings.diMag3RemoteClampOpenCtrl > 0 AND g_tyNtParamCurr.tyDOSettings.diMag3RemoteClampOpenCtrl <= UDINT_TO_DINT(c_udiDOutputMax) THEN
		a_bPhysicalDO[g_tyNtParamCurr.tyDOSettings.diMag3RemoteClampOpenCtrl]	:= NOT  p_bMag3RemoteClampOpenCtrl;
	END_IF

	IF g_tyNtParamCurr.tyDOSettings.diBypCurtainSen > 0 AND g_tyNtParamCurr.tyDOSettings.diBypCurtainSen <= UDINT_TO_DINT(c_udiDOutputMax) THEN
		a_bPhysicalDO[g_tyNtParamCurr.tyDOSettings.diBypCurtainSen]	:= p_bBypCurtainSen;
	END_IF

	IF g_tyNtParamCurr.tyDOSettings.diRstCurtainSen > 0 AND g_tyNtParamCurr.tyDOSettings.diRstCurtainSen <= UDINT_TO_DINT(c_udiDOutputMax) THEN
		a_bPhysicalDO[g_tyNtParamCurr.tyDOSettings.diRstCurtainSen]	:= p_bRstCurtainSen;
	END_IF

	IF g_tyNtParamCurr.tyDOSettings.diBypCurtainPBLED > 0 AND g_tyNtParamCurr.tyDOSettings.diBypCurtainPBLED <= UDINT_TO_DINT(c_udiDOutputMax) THEN
		a_bPhysicalDO[g_tyNtParamCurr.tyDOSettings.diBypCurtainPBLED]	:= p_bBypCurtainPBLED;
	END_IF

	IF g_tyNtParamCurr.tyDOSettings.diScanTrigSig > 0 AND g_tyNtParamCurr.tyDOSettings.diScanTrigSig <= UDINT_TO_DINT(c_udiDOutputMax) THEN
		a_bPhysicalDO[g_tyNtParamCurr.tyDOSettings.diScanTrigSig]	:= p_bScanTrigSig;
	END_IF

	IF g_tyNtParamCurr.tyDOSettings.diMag1ExitPCB > 0 AND g_tyNtParamCurr.tyDOSettings.diMag1ExitPCB <= UDINT_TO_DINT(c_udiDOutputMax) THEN
		a_bPhysicalDO[g_tyNtParamCurr.tyDOSettings.diMag1ExitPCB]	:= p_bMag1ExitPCB;
	END_IF

	IF g_tyNtParamCurr.tyDOSettings.diMag2ExitPCB > 0 AND g_tyNtParamCurr.tyDOSettings.diMag2ExitPCB <= UDINT_TO_DINT(c_udiDOutputMax) THEN
		a_bPhysicalDO[g_tyNtParamCurr.tyDOSettings.diMag2ExitPCB]	:= p_bMag2ExitPCB;
	END_IF

	IF g_tyNtParamCurr.tyDOSettings.diMag3ExitPCB > 0 AND g_tyNtParamCurr.tyDOSettings.diMag3ExitPCB <= UDINT_TO_DINT(c_udiDOutputMax) THEN
		a_bPhysicalDO[g_tyNtParamCurr.tyDOSettings.diMag3ExitPCB]	:= p_bMag3ExitPCB;
	END_IF

	//Update Output
	g_tyDOutput.bSafetyRlyRst			:= a_bPhysicalDO[g_tyNtParamCurr.tyDOSettings.diSafetyRlyRst];
	g_tyDOutput.bTLRed					:= a_bPhysicalDO[g_tyNtParamCurr.tyDOSettings.diTLRed];
	g_tyDOutput.bTLAmber				:= a_bPhysicalDO[g_tyNtParamCurr.tyDOSettings.diTLAmber];
	g_tyDOutput.bTLGreen				:= a_bPhysicalDO[g_tyNtParamCurr.tyDOSettings.diTLGreen];
	g_tyDOutput.bBuzzer					:= a_bPhysicalDO[g_tyNtParamCurr.tyDOSettings.diBuzzer];
	g_tyDOutput.bUSBA					:= a_bPhysicalDO[g_tyNtParamCurr.tyDOSettings.diUSBA];
	g_tyDOutput.bUSBB					:= a_bPhysicalDO[g_tyNtParamCurr.tyDOSettings.diUSBB];
	g_tyDOutput.bOvenInfoSigA			:= a_bPhysicalDO[g_tyNtParamCurr.tyDOSettings.diOvenInfoSigA];
	g_tyDOutput.bOvenInfoSigB			:= a_bPhysicalDO[g_tyNtParamCurr.tyDOSettings.diOvenInfoSigB];
	g_tyDOutput.bPusherExtCtrl			:= a_bPhysicalDO[g_tyNtParamCurr.tyDOSettings.diPusherExtCtrl];
	g_tyDOutput.bStopperUnBlkCtrlA		:= a_bPhysicalDO[g_tyNtParamCurr.tyDOSettings.diStopperUnblkCtrlA];
	g_tyDOutput.bStopperUnBlkCtrlB		:= a_bPhysicalDO[g_tyNtParamCurr.tyDOSettings.diStopperUnblkCtrlB];
	g_tyDOutput.bMag1FixedClampCtrl		:= a_bPhysicalDO[g_tyNtParamCurr.tyDOSettings.diMag1FixedClampCtrl];
	g_tyDOutput.bMag1RemoteClampCtrl	:= a_bPhysicalDO[g_tyNtParamCurr.tyDOSettings.diMag1RemoteClampCtrl];
	g_tyDOutput.bMag2FixedClampCtrl		:= a_bPhysicalDO[g_tyNtParamCurr.tyDOSettings.diMag2FixedClampCtrl];
	g_tyDOutput.bMag2RemoteClampCtrl	:= a_bPhysicalDO[g_tyNtParamCurr.tyDOSettings.diMag2RemoteClampCtrl];
	g_tyDOutput.bMag3FixedClampCtrl		:= a_bPhysicalDO[g_tyNtParamCurr.tyDOSettings.diMag3FixedClampCtrl];
	g_tyDOutput.bMag3RemoteClampCtrl	:= a_bPhysicalDO[g_tyNtParamCurr.tyDOSettings.diMag3RemoteClampCtrl];
	g_tyDOutput.bInShutterOpenCtrl		:= a_bPhysicalDO[g_tyNtParamCurr.tyDOSettings.diInShutterOpenCtrl];
	g_tyDOutput.bInShutterCloseCtrl		:= a_bPhysicalDO[g_tyNtParamCurr.tyDOSettings.diInShutterCloseCtrl];
	g_tyDOutput.bOutShutterOpenCtrl		:= a_bPhysicalDO[g_tyNtParamCurr.tyDOSettings.diOutShutterOpenCtrl];
	g_tyDOutput.bOutShutterCloseCtrl	:= a_bPhysicalDO[g_tyNtParamCurr.tyDOSettings.diOutShutterCloseCtrl];
	g_tyDOutput.bMag1ConvMtrIn			:= a_bPhysicalDO[g_tyNtParamCurr.tyDOSettings.diMag1ConvMtrIn];
	g_tyDOutput.bMag1ConvMtrOut			:= a_bPhysicalDO[g_tyNtParamCurr.tyDOSettings.diMag1ConvMtrOut];
	g_tyDOutput.bMag2ConvMtrIn			:= a_bPhysicalDO[g_tyNtParamCurr.tyDOSettings.diMag2ConvMtrIn];
	g_tyDOutput.bMag2ConvMtrOut			:= a_bPhysicalDO[g_tyNtParamCurr.tyDOSettings.diMag2ConvMtrOut];
	g_tyDOutput.bMag3ConvMtrIn			:= a_bPhysicalDO[g_tyNtParamCurr.tyDOSettings.diMag3ConvMtrIn];
	g_tyDOutput.bMag3ConvMtrOut			:= a_bPhysicalDO[g_tyNtParamCurr.tyDOSettings.diMag3ConvMtrOut];
	g_tyDOutput.bMag1SelClampCtrl		:= a_bPhysicalDO[g_tyNtParamCurr.tyDOSettings.diMag1SelClampCtrl];
	g_tyDOutput.bMag2SelClampCtrl		:= a_bPhysicalDO[g_tyNtParamCurr.tyDOSettings.diMag2SelClampCtrl];
	g_tyDOutput.bMag3SelClampCtrl		:= a_bPhysicalDO[g_tyNtParamCurr.tyDOSettings.diMag3SelClampCtrl];
	g_tyDOutput.bMag1SelUnClampCtrl		:= a_bPhysicalDO[g_tyNtParamCurr.tyDOSettings.diMag1SelUnclampCtrl];
	g_tyDOutput.bMag2SelUnClampCtrl		:= a_bPhysicalDO[g_tyNtParamCurr.tyDOSettings.diMag2SelUnclampCtrl];
	g_tyDOutput.bMag3SelUnClampCtrl		:= a_bPhysicalDO[g_tyNtParamCurr.tyDOSettings.diMag3SelUnclampCtrl];
	g_tyDOutput.bPusherConvMtrOn		:= a_bPhysicalDO[g_tyNtParamCurr.tyDOSettings.diPushConvMtrOn];
	g_tyDOutput.bMag1WallEngageCtrl		:= a_bPhysicalDO[g_tyNtParamCurr.tyDOSettings.diMag1WallEngageCtrl];
	g_tyDOutput.bMag2WallEngageCtrl		:= a_bPhysicalDO[g_tyNtParamCurr.tyDOSettings.diMag2WallEngageCtrl];
	g_tyDOutput.bMag3WallEngageCtrl		:= a_bPhysicalDO[g_tyNtParamCurr.tyDOSettings.diMag3WallEngageCtrl];
	g_tyDOutput.bMag1SafetyBarRetCtrl	:= a_bPhysicalDO[g_tyNtParamCurr.tyDOSettings.diMag1SafetyBarRetCtrl];
	g_tyDOutput.bMag2SafetyBarRetCtrl	:= a_bPhysicalDO[g_tyNtParamCurr.tyDOSettings.diMag2SafetyBarRetCtrl];
	g_tyDOutput.bMag3SafetyBarRetCtrl	:= a_bPhysicalDO[g_tyNtParamCurr.tyDOSettings.diMag3SafetyBarRetCtrl];
	g_tyDOutput.bSOT1MagAvailable		:= a_bPhysicalDO[g_tyNtParamCurr.tyDOSettings.diSOT1MagAvailable];
	g_tyDOutput.bSOT2MagAvailable		:= a_bPhysicalDO[g_tyNtParamCurr.tyDOSettings.diSOT2MagAvailable];
	g_tyDOutput.bSOT3MagAvailable		:= a_bPhysicalDO[g_tyNtParamCurr.tyDOSettings.diSOT3MagAvailable];
	g_tyDOutput.bSOT4MagAvailable		:= a_bPhysicalDO[g_tyNtParamCurr.tyDOSettings.diSOT4MagAvailable];
	g_tyDOutput.bSOT1MagError			:= a_bPhysicalDO[g_tyNtParamCurr.tyDOSettings.diSOT1MagError];
	g_tyDOutput.bSOT2MagError			:= a_bPhysicalDO[g_tyNtParamCurr.tyDOSettings.diSOT2MagError];
	g_tyDOutput.bSOT3MagError			:= a_bPhysicalDO[g_tyNtParamCurr.tyDOSettings.diSOT3MagError];
	g_tyDOutput.bSOT4MagError			:= a_bPhysicalDO[g_tyNtParamCurr.tyDOSettings.diSOT4MagError];
	g_tyDOutput.bSOT1MagReady			:= a_bPhysicalDO[g_tyNtParamCurr.tyDOSettings.diSOT1MagReady];
	g_tyDOutput.bSOT2MagReady			:= a_bPhysicalDO[g_tyNtParamCurr.tyDOSettings.diSOT2MagReady];
	g_tyDOutput.bSOT3MagReady			:= a_bPhysicalDO[g_tyNtParamCurr.tyDOSettings.diSOT3MagReady];
	g_tyDOutput.bSOT4MagReady			:= a_bPhysicalDO[g_tyNtParamCurr.tyDOSettings.diSOT4MagReady];
	g_tyDOutput.bSOT1MagSizeLarge		:= a_bPhysicalDO[g_tyNtParamCurr.tyDOSettings.diSOTMagSizeLarge1];
	g_tyDOutput.bSOT2MagSizeLarge		:= a_bPhysicalDO[g_tyNtParamCurr.tyDOSettings.diSOTMagSizeLarge2];
	g_tyDOutput.bSOT3MagSizeLarge		:= a_bPhysicalDO[g_tyNtParamCurr.tyDOSettings.diSOTMagSizeLarge3];
	g_tyDOutput.bSOT4MagSizeLarge		:= a_bPhysicalDO[g_tyNtParamCurr.tyDOSettings.diSOTMagSizeLarge4];
	g_tyDOutput.bMagAWOpenLimByp1		:= a_bPhysicalDO[g_tyNtParamCurr.tyDOSettings.diMagAWOpenLimByp1];
	g_tyDOutput.bMagAWOpenLimByp2		:= a_bPhysicalDO[g_tyNtParamCurr.tyDOSettings.diMagAWOpenLimByp2];
	g_tyDOutput.bMagAWOpenLimByp3		:= a_bPhysicalDO[g_tyNtParamCurr.tyDOSettings.diMagAWOpenLimByp3];
	g_tyDOutput.bMagAWOpenLimByp4		:= a_bPhysicalDO[g_tyNtParamCurr.tyDOSettings.diMagAWOpenLimByp4];
	g_tyDOutput.bMagAWSmallLimSen1		:= a_bPhysicalDO[g_tyNtParamCurr.tyDOSettings.diMagAWSmallLimSen1];
	g_tyDOutput.bMagAWSmallLimSen2		:= a_bPhysicalDO[g_tyNtParamCurr.tyDOSettings.diMagAWSmallLimSen2];
	g_tyDOutput.bMagAWSmallLimSen3		:= a_bPhysicalDO[g_tyNtParamCurr.tyDOSettings.diMagAWSmallLimSen3];
	g_tyDOutput.bMagAWSmallLimSen4		:= a_bPhysicalDO[g_tyNtParamCurr.tyDOSettings.diMagAWSmallLimSen4];
	g_tyDOutput.bMag1ReqToBring			:= a_bPhysicalDO[g_tyNtParamCurr.tyDOSettings.diMag1ReqToBring];
	g_tyDOutput.bMag1ReqToGet			:= a_bPhysicalDO[g_tyNtParamCurr.tyDOSettings.diMag1ReqToGet];
	g_tyDOutput.bMag2ReqToBring			:= a_bPhysicalDO[g_tyNtParamCurr.tyDOSettings.diMag2ReqToBring];
	g_tyDOutput.bMag2ReqToGet			:= a_bPhysicalDO[g_tyNtParamCurr.tyDOSettings.diMag2ReqToGet];
	g_tyDOutput.bMag3ReqToBring			:= a_bPhysicalDO[g_tyNtParamCurr.tyDOSettings.diMag3ReqToBring];
	g_tyDOutput.bMag3ReqToGet			:= a_bPhysicalDO[g_tyNtParamCurr.tyDOSettings.diMag3ReqToGet];
	g_tyDOutput.bMag4ReqToBring			:= a_bPhysicalDO[g_tyNtParamCurr.tyDOSettings.diMag4ReqToBring];
	g_tyDOutput.bMag4ReqToGet			:= a_bPhysicalDO[g_tyNtParamCurr.tyDOSettings.diMag4ReqToGet];
	g_tyDOutput.bMtrPshrExt				:= a_bPhysicalDO[g_tyNtParamCurr.tyDOSettings.diMtrPshrExt];
	g_tyDOutput.bMtrPshrRet				:= a_bPhysicalDO[g_tyNtParamCurr.tyDOSettings.diMtrPshrRet];
	g_tyDOutput.bMtrPshrOn				:= a_bPhysicalDO[g_tyNtParamCurr.tyDOSettings.diMtrPshrOn];
	g_tyDOutput.bMtrPshrBrakeRls		:= a_bPhysicalDO[g_tyNtParamCurr.tyDOSettings.diMtrPshrBrakeRls];
	g_tyDOutput.bMtrPshrSpdBinBit0		:= a_bPhysicalDO[g_tyNtParamCurr.tyDOSettings.diMtrPshrSpdBinBit0];
	g_tyDOutput.bMtrPshrSpdBinBit1		:= a_bPhysicalDO[g_tyNtParamCurr.tyDOSettings.diMtrPshrSpdBinBit1];
	g_tyDOutput.bMtrPshrSpdBinBit2		:= a_bPhysicalDO[g_tyNtParamCurr.tyDOSettings.diMtrPshrSpdBinBit2];
	g_tyDOutput.bMtrPshrAlmRst			:= a_bPhysicalDO[g_tyNtParamCurr.tyDOSettings.diMtrPshrAlmRst];
	IF a_bPhysicalDO[g_tyNtParamCurr.tyDOSettings.diLinkProjMagConvLane1Prep THEN
		g_tyDOutput.bEntTopStprUnblkCtrl	:= a_bPhysicalDO[g_tyNtParamCurr.tyDOSettings.diEntTopStprUnblkCtrl];
		g_tyDOutput.bMidTopStprUnblkCtrl	:= a_bPhysicalDO[g_tyNtParamCurr.tyDOSettings.diMidTopStprUnblkCtrl];
		g_tyDOutput.bExtTopStprUnblkCtrl	:= a_bPhysicalDO[g_tyNtParamCurr.tyDOSettings.diExtTopStprUnblkCtrl];
		g_tyDOutput.bMidBtmStprUnblkCtrl	:= a_bPhysicalDO[g_tyNtParamCurr.tyDOSettings.diMidBtmStprUnblkCtrl];
		g_tyDOutput.bExtBtmStprUnblkCtrl	:= a_bPhysicalDO[g_tyNtParamCurr.tyDOSettings.diExtBtmStprUnblkCtrl];
	END_IF
	IF a_bPhysicalDO[g_tyNtParamCurr.tyDOSettings.diLinkProjMagConvLane1Prep THEN
		g_tyDOutput.bEntTopStprUnblkCtrl2	:= a_bPhysicalDO[g_tyNtParamCurr.tyDOSettings.diEntTopStprUnblkCtrl2];
		g_tyDOutput.bMidTopStprUnblkCtrl2	:= a_bPhysicalDO[g_tyNtParamCurr.tyDOSettings.diMidTopStprUnblkCtrl2];
		g_tyDOutput.bExtTopStprUnblkCtrl2	:= a_bPhysicalDO[g_tyNtParamCurr.tyDOSettings.diExtTopStprUnblkCtrl2];
		g_tyDOutput.bMidBtmStprUnblkCtrl2	:= a_bPhysicalDO[g_tyNtParamCurr.tyDOSettings.diMidBtmStprUnblkCtrl2];
		g_tyDOutput.bExtBtmStprUnblkCtrl2	:= a_bPhysicalDO[g_tyNtParamCurr.tyDOSettings.diExtBtmStprUnblkCtrl2];
	END_IF
	g_tyDOutput.bMtrPwrRly			:= a_bPhysicalDO[g_tyNtParamCurr.tyDOSettings.diMtrPwrRly];

	g_tyDOutput.bMag1FixedClampOpenCtrl		:= a_bPhysicalDO[g_tyNtParamCurr.tyDOSettings.diMag1FixedClampOpenCtrl];
	g_tyDOutput.bMag1RemoteClampOpenCtrl	:= a_bPhysicalDO[g_tyNtParamCurr.tyDOSettings.diMag1RemoteClampOpenCtrl];
	g_tyDOutput.bMag2FixedClampOpenCtrl		:= a_bPhysicalDO[g_tyNtParamCurr.tyDOSettings.diMag2FixedClampOpenCtrl];
	g_tyDOutput.bMag2RemoteClampOpenCtrl	:= a_bPhysicalDO[g_tyNtParamCurr.tyDOSettings.diMag2RemoteClampOpenCtrl];
	g_tyDOutput.bMag3FixedClampOpenCtrl		:= a_bPhysicalDO[g_tyNtParamCurr.tyDOSettings.diMag3FixedClampOpenCtrl];
	g_tyDOutput.bMag3RemoteClampOpenCtrl	:= a_bPhysicalDO[g_tyNtParamCurr.tyDOSettings.diMag3RemoteClampOpenCtrl];

	g_tyDOutput.bOutShutterOpenCtrl2		:= a_bPhysicalDO[g_tyNtParamCurr.tyDOSettings.diOutShutterOpenCtrl2];
	g_tyDOutput.bOutShutterCloseCtrl2		:= a_bPhysicalDO[g_tyNtParamCurr.tyDOSettings.diOutShutterCloseCtrl2];

	g_tyDOutput.bOutShutterOpenCtrl3		:= a_bPhysicalDO[g_tyNtParamCurr.tyDOSettings.diOutShutterOpenCtrl3];
	g_tyDOutput.bOutShutterCloseCtrl3		:= a_bPhysicalDO[g_tyNtParamCurr.tyDOSettings.diOutShutterCloseCtrl3];

	g_tyDOutput.bBypCurtainSen				:= a_bPhysicalDO[g_tyNtParamCurr.tyDOSettings.diBypCurtainSen];
	g_tyDOutput.bRstCurtainSen				:= a_bPhysicalDO[g_tyNtParamCurr.tyDOSettings.diRstCurtainSen];
	g_tyDOutput.bBypCurtainPBLED			:= a_bPhysicalDO[g_tyNtParamCurr.tyDOSettings.diBypCurtainPBLED];

	g_tyDOutput.diMag1ExitPCB				:=	a_bPhysicalDO[g_tyNtParamCurr.tyDOSettings.diMag1ExitPCB];
	g_tyDOutput.diMag2ExitPCB 				:= 	a_bPhysicalDO[g_tyNtParamCurr.tyDOSettings.diMag2ExitPCB];
	g_tyDOutput.diMag3ExitPCB 				:=	a_bPhysicalDO[g_tyNtParamCurr.tyDOSettings.diMag3ExitPCB];
	g_tyDOutput.diScanTrigSig				:=	a_bPhysicalDO[g_tyNtParamCurr.tyDOSettings.diScanTrigSig];
END_ACTION
```

#### Local.var - Change By Project
```iecst
(*2019-04-30*)
(**)
(*Local Action, State & Status*)
VAR
	eAct : eDOAction := DOActIdle;
	eStat : eDOAction := DOActIdle;
	eStatus : eFBStatus := Idle;
	sStatTxt : STRING[200] := '';
	a_sStatText : ARRAY[0..50] OF STRING[200] := ['Idling','Resetting All Special Output','Turning On Bypass Cover Switch','Turning Off Bypass Cover Switch',47('')];
END_VAR
(**)
(*Local Alarm*)
(**)
(*Local Output*)
VAR
	tyDOutput : tyDigitalOutput;
END_VAR
(**)
(*Local Input*)
VAR
	tyDOSettings : tyDigitalOutputSettings;
END_VAR
(**)
VAR
	bManual : BOOL := FALSE;
END_VAR
(**)
(*Local*)
VAR
	bInitDone : BOOL;
	bInitialDone : BOOL;
	a_bPhysicalDO : ARRAY[1..c_udiDOutputMax] OF BOOL;
	eStatOld : eDOAction := DOActIdle;
	usiShutterTuningStep : USINT := 0;
	bShutterTuning : BOOL;
	fbShutterTuneOpnTim : TON := (PT:=T#2s);
	fbShutterTuneClsTim : TON := (PT:=T#2s);
	bAgvComIODisabled : BOOL;
END_VAR
(*Link*)
VAR
	bSOTMagError1 : BOOL;
	bSOTMagSLarge1 : BOOL;
	bSOTMagReady1 : BOOL;
	bSOTMagAvailable1 : BOOL;
	bSOTMagError2 : BOOL;
	bSOTMagSLarge2 : BOOL;
	bSOTMagReady2 : BOOL;
	bSOTMagAvailable2 : BOOL;
	bSOTMagError3 : BOOL;
	bSOTMagSLarge3 : BOOL;
	bSOTMagReady3 : BOOL;
	bSOTMagAvailable3 : BOOL;
	bSOTMagError4 : BOOL;
	bSOTMagSLarge4 : BOOL;
	bSOTMagReady4 : BOOL;
	bSOTMagAvailable4 : BOOL;
	bRequestToBring1 : BOOL;
	bRequestToGet1 : BOOL;
	bRequestToBring2 : BOOL;
	bRequestToGet2 : BOOL;
	bRequestToBring3 : BOOL;
	bRequestToGet3 : BOOL;
	bRequestToBring4 : BOOL;
	bRequestToGet4 : BOOL;
	bBypCurtainSen : BOOL;
	bRstCurtainSen : BOOL;
	bBypCurtainPBLED : BOOL;
	bMagAWOpenLimByp1 : BOOL;
	bMagAWOpenLimByp2 : BOOL;
	bMagAWOpenLimByp3 : BOOL;
	bMagAWOpenLimByp4 : BOOL;
	bMagAWSmallLimSen1 : BOOL;
	bMagAWSmallLimSen2 : BOOL;
	bMagAWSmallLimSen3 : BOOL;
	bMagAWSmallLimSen4 : BOOL;
	bScanTrigSig : BOOL;
	bMag1ExitPCB : BOOL;
	bMag2ExitPCB : BOOL;
	bMag3ExitPCB : BOOL;
END_VAR
```

#### Act_InitGlobal.st - Change By Project
```iecst
(** 2019-05-20 **)
ACTION Act_InitGlobal:

	(* Always Change If Project Change *)

	//Pass Data To Link
	p_bLinkStartupRun ACCESS p_StartupRun;
	p_bLinkOpsRun ACCESS p_OpsRun;
	p_bLinkError ACCESS p_AlarmErr;
	p_eLinkAGVComProtocol ACCESS p_McParamAGVComProtocol;
	p_bLinkNtParamProjSOTSenPrep ACCESS p_NtParamProjSOTSenPrep;
	p_bLinkProjMagConvLane1Prep ACCESS p_NtParamProjMagConvLane1Prep;
	p_bLinkProjMagConvLane2Prep ACCESS p_NtParamProjMagConvLane2Prep;

	p_bLinkAGVCommRdy1 ACCESS p_OpsAGVCommRdy1;
	p_bLinkAGVCommRdy2 ACCESS p_OpsAGVCommRdy2;
	p_bLinkAGVCommRdy3 ACCESS p_OpsAGVCommRdy3;

	p_bLinkOpsBypCurtainLED ACCESS p_OpsTravLifULBypCurtainLED;	//Bypass Curtain Push Button LED
	p_bLinkOpsBypCurtainSen ACCESS p_OpsTravLifULBypCurtainSenCtrl; //Bypass the Curtain Sensor

	//Pass Data To Internal Use
	p_eAct ACCESS p_UIDOAct;
	p_tyDOSettings ACCESS p_NtParamDOSettings;
	p_bManual ACCESS p_UIUIMnlMod;
	p_bSafetyRlyRst ACCESS p_RstErrSafetyRlyRst;
	p_bTLRed ACCESS p_TLBuzRed;
	p_bTLAmber ACCESS p_TLBuzAmber;
	p_bTLGreen ACCESS p_TLBuzGreen;
	p_bBuzzer ACCESS p_TLBuzBeep;
	p_bUSBA ACCESS p_USSMEMAAUSB;
	p_bUSBB ACCESS p_USSMEMABUSB;
	p_bOvenInfoSigA ACCESS p_OvenInfoAOvenAllow;
	p_bOvenInfoSigB ACCESS p_OvenInfoBOvenAllow;
	p_bPusherExtCtrl ACCESS p_PshrConvPshrExtCtrl;
	p_bStopperUnblkCtrlA ACCESS p_PneuNoSenStopperARetCtrl;
	p_bStopperUnblkCtrlB ACCESS p_PneuNoSenStopperBRetCtrl;
//	p_bMag1FixedClampCtrl ACCESS p_MagConv2Clp1FixClprClampCtrl; //share lifter mag clmp -act_link
	p_bMag1RemoteClampCtrl ACCESS p_MagConv2Clp1RmtClprClampCtrl;
//	p_bMag2FixedClampCtrl ACCESS p_MagConv2Clp2FixClprClampCtrl;
	p_bMag2RemoteClampCtrl ACCESS p_MagConv2Clp2RmtClprClampCtrl;
	p_bMag3FixedClampCtrl ACCESS p_MagConv2Clp3FixClprClampCtrl;
	p_bMag3RemoteClampCtrl ACCESS p_MagConv2Clp3RmtClprClampCtrl;
	p_bInShutterOpenCtrl ACCESS p_Pneu2SenInShutterRetCtrl;
	p_bInShutterCloseCtrl ACCESS p_Pneu2SenInShutterExtCtrl;
	p_bOutShutterOpenCtrl ACCESS p_Pneu2SenOutShutterRetCtrl;
	p_bOutShutterCloseCtrl ACCESS p_Pneu2SenOutShutterExtCtrl;
//	p_bMag1ConvMtrIn ACCESS p_MagConv2Clp1MtrSigOnOrLToR; //share lifter mag conv -act_link
//	p_bMag1ConvMtrOut ACCESS p_MagConv2Clp1MtrDirOrRToL;
//	p_bMag2ConvMtrIn ACCESS p_MagConv2Clp2MtrSigOnOrLToR;
//	p_bMag2ConvMtrOut ACCESS p_MagConv2Clp2MtrDirOrRToL;
	p_bMag3ConvMtrIn ACCESS p_MagConv2Clp3MtrSigOnOrLToR;
	p_bMag3ConvMtrOut ACCESS p_MagConv2Clp3MtrDirOrRToL;
	p_bMag1SelClampCtrl ACCESS p_PneuNoSenSelClamp1RetCtrl;
	p_bMag2SelClampCtrl ACCESS p_PneuNoSenSelClamp2RetCtrl;
	p_bMag3SelClampCtrl ACCESS p_PneuNoSenSelClamp3RetCtrl;
	p_bMag1SelUnclampCtrl ACCESS p_PneuNoSenSelClamp1ExtCtrl;
	p_bMag2SelUnclampCtrl ACCESS p_PneuNoSenSelClamp2ExtCtrl;
	p_bMag3SelUnclampCtrl ACCESS p_PneuNoSenSelClamp3ExtCtrl;

	p_bPushConvMtrOn ACCESS p_PshrConvMtrSigOnOrLToR;
	p_bMag1WallEngageCtrl ACCESS p_Pneu2SMag1AWEngageExtCtrl;
	p_bMag2WallEngageCtrl ACCESS p_Pneu2SMag2AWEngageExtCtrl;
	p_bMag3WallEngageCtrl ACCESS p_Pneu2SMag3AWEngageExtCtrl;
	p_bMag1SafetyBarRetCtrl ACCESS p_Pneu2SMag1SafetyBarRetCtrl;
	p_bMag2SafetyBarRetCtrl ACCESS p_Pneu2SMag2SafetyBarRetCtrl;
	p_bMag3SafetyBarRetCtrl ACCESS p_Pneu2SMag3SafetyBarRetCtrl;
	p_bMtrPshrExt ACCESS p_MtrPshrCW;
	p_bMtrPshrRet ACCESS p_MtrPshrCCW;
	p_bMtrPshrOn ACCESS p_MtrPshrSigOn;
	p_bMtrPshrBrakeRls ACCESS p_MtrPshrBrake;
	p_bMtrPshrSpdBinBit0 ACCESS p_MtrPshrSpdBinBit0;
	p_bMtrPshrSpdBinBit1 ACCESS p_MtrPshrSpdBinBit1;
	p_bMtrPshrSpdBinBit2 ACCESS p_MtrPshrSpdBinBit2;
	p_bMtrPshrAlmRst ACCESS p_MtrPshrAlmRst;

	p_bEntTopStprUnblkCtrl ACCESS p_PneuNoSenTopEntStprRetCtrl;
	p_bMidTopStprUnblkCtrl ACCESS p_PneuNoSenTopMidStprExtCtrl;
	p_bExtTopStprUnblkCtrl ACCESS p_PneuNoSenTopExtStprRetCtrl;
	p_bMidBtmStprUnblkCtrl ACCESS p_PneuNoSenBtmMidStprExtCtrl;
	p_bExtBtmStprUnblkCtrl ACCESS p_PneuNoSenBtmExtStprRetCtrl;
	p_bEntTopStprUnblkCtrl2 ACCESS p_PneuNoSenTopEntStpr2RetCtrl;
	p_bMidTopStprUnblkCtrl2 ACCESS p_PneuNoSenTopMidStpr2ExtCtrl;
	p_bExtTopStprUnblkCtrl2 ACCESS p_PneuNoSenTopExtStpr2RetCtrl;
	p_bMidBtmStprUnblkCtrl2 ACCESS p_PneuNoSenBtmMidStpr2ExtCtrl;
	p_bExtBtmStprUnblkCtrl2 ACCESS p_PneuNoSenBtmExtStpr2RetCtrl;
	p_bInMagConvMtrOn ACCESS p_InMagConvMtrDirOrRToL;
	p_bOutMagConvMtrOn ACCESS p_OutMagConvMtrSigOnOrLToR;
	p_bInMagConv2MtrOn ACCESS p_InMagConv2MtrDirOrRToL;
	p_bOutMagConv2MtrOn ACCESS p_OutMagConv2MtrSigOnOrLToR;

	p_bMag1FixedClampOpenCtrl ACCESS p_MagConv2Clp1FixClprClampCtrl;
	p_bMag1RemoteClampOpenCtrl ACCESS p_MagConv2Clp1RmtClprClampCtrl;
	p_bMag2FixedClampOpenCtrl ACCESS p_MagConv2Clp2FixClprClampCtrl;
	p_bMag2RemoteClampOpenCtrl ACCESS p_MagConv2Clp2RmtClprClampCtrl;
	p_bMag3FixedClampOpenCtrl ACCESS p_MagConv2Clp3FixClprClampCtrl;
	p_bMag3RemoteClampOpenCtrl ACCESS p_MagConv2Clp3RmtClprClampCtrl;

	p_bOutShutterOpenCtrl2 ACCESS p_Pneu2SenOutShutterRetCtrl2;
	p_bOutShutterCloseCtrl2 ACCESS p_Pneu2SenOutShutterExtCtrl2;
	p_bOutShutterOpenCtrl3 ACCESS p_Pneu2SenOutShutterRetCtrl3;
	p_bOutShutterCloseCtrl3 ACCESS p_Pneu2SenOutShutterExtCtrl3;

	p_bInletStopperExtCtrl ACCESS p_InletStopperExtCtrl;
	p_bInletStopperRetCtrl ACCESS p_InletStopperRetCtrl;

	p_eCustomerReq ACCESS p_NtParamCustomerReq;
	(* Always Change If Project Change *)

END_ACTION
```

#### InputRef_Link.var - Change By Project
```iecst
(*2021-05-25*)
(**)
(*General*)
VAR
	p_bLinkStartupRun : REFERENCE TO BOOL;
	p_bLinkOpsRun : REFERENCE TO BOOL;
	p_bLinkError : REFERENCE TO BOOL;
	p_eLinkAGVComProtocol : REFERENCE TO eMcAGVCommProtocol;
	p_bLinkNtParamProjSOTSenPrep : REFERENCE TO BOOL;
	p_bLinkProjMagConvLane1Prep : REFERENCE TO BOOL;
	p_bLinkProjMagConvLane2Prep : REFERENCE TO BOOL;
	p_bLinkAGVCommRdy1 : REFERENCE TO BOOL;
	p_bLinkAGVCommRdy2 : REFERENCE TO BOOL;
	p_bLinkAGVCommRdy3 : REFERENCE TO BOOL;
	p_bLinkOpsBypCurtainSen : REFERENCE TO BOOL;
	p_bLinkOpsBypCurtainLED : REFERENCE TO BOOL;
END_VAR
```

#### Act_Link.st - Change By Project
```iecst
(** 2019-05-20 **)
ACTION Act_Link:
	//
	IF p_eCustomerReq = Siemens THEN
		bTLAmber := g_tyTLBuzWhite;
	ELSE
		bTLAmber := g_tyTLBuzAmber;
	END_IF

	//Motor power relay
	IF bLinkStartupRun = FALSE THEN
		bMtrPwrRly		:= TRUE;
	END_IF

	IF g_tyUIOut.bManualMod THEN

		bSOTMagError1	:= g_tyUISOTMagErr1;
		bSOTMagError2	:= g_tyUISOTMagErr2;
		bSOTMagError3	:= g_tyUISOTMagErr3;
		//		bSOTMagError4	:= g_tyUISOTMagErr4;
		bSOTMagReady1	:= g_tyUISOTMagRdy1;
		bSOTMagReady2	:= g_tyUISOTMagRdy2;
		bSOTMagReady3	:= g_tyUISOTMagRdy3;
		//		bSOTMagReady4	:= g_tyUISOTMagRdy4;
		bSOTMagAvailable1	:= g_tyUISOTMagAvail1;
		bSOTMagAvailable2	:= g_tyUISOTMagAvail2;
		bSOTMagAvailable3	:= g_tyUISOTMagAvail3;
		//		bSOTMagAvailable4	:= g_tyUISOTMagAvail4;
		bSOTMagSizeLarge1	:= g_tyUISOTMagSLarge1;
		bSOTMagSizeLarge2	:= g_tyUISOTMagSLarge2;
		bSOTMagSizeLarge3 := g_tyUISOTMagSLarge3;
		//		bSOTMagSizeLarge4	:= g_tyUISOTMagSLarge4;

		bMagAWOpenLimByp1 := g_tyUIMagAWOpenLimByp1;
		bMagAWOpenLimByp2 := g_tyUIMagAWOpenLimByp2;
		bMagAWOpenLimByp3 := g_tyUIMagAWOpenLimByp3;
		//		bMagAWOpenLimByp4 := g_tyUIMagAWOpenLimByp4;

		bMagAWSmallLimSen1 := g_tyUIMagAWSmallLimSen1;
		bMagAWSmallLimSen2 := g_tyUIMagAWSmallLimSen2;
		bMagAWSmallLimSen3 := g_tyUIMagAWSmallLimSen3;
		//		bMagAWSmallLimSen4 := g_tyUIMagAWSmallLimSen4;

		bRequestToBring1 := g_tyUIAIVReqBring1;
		bRequestToBring2 := g_tyUIAIVReqBring2;
		bRequestToBring3 := g_tyUIAIVReqBring3;

		bRequestToGet1 := g_tyUIAIVReqGet1;
		bRequestToGet2 := g_tyUIAIVReqGet2;
		bRequestToGet3 := g_tyUIAIVReqGet3;

		//DMCRFID
		bScanTrigSig := g_tyUIStartScanSig;
		bMag1ExitPCB := g_tyUIMag1TransOut;
		bMag2ExitPCB := g_tyUIMag2TransOut;
		bMag3ExitPCB := g_tyUIMag3TransOut;

	ELSIF g_tyOps.bRun THEN
		bSOTMagReady1 := g_tyUSSOT1USB;
		bSOTMagReady2 := g_tyUSSOT2USB;
		bSOTMagReady3 := g_tyUSSOT3USB;

		bSOTMagError1 := g_tyAlarmErr;
		bSOTMagError2 := g_tyAlarmErr;
		bSOTMagError3 := g_tyAlarmErr;

		bSOTMagAvailable1 := g_tyDSSOT1DBA;
		bSOTMagAvailable2 := g_tyDSSOT2DBA;
		bSOTMagAvailable3 := g_tyDSSOT3DBA;

		bSOTMagSizeLarge1 := g_tyDSSOT1MagSizeLarge;
		bSOTMagSizeLarge2 := g_tyDSSOT2MagSizeLarge;
		bSOTMagSizeLarge3 := g_tyDSSOT3MagSizeLarge;

		bRequestToBring1 := g_tyBuffer1MagRemoved;
		bRequestToBring2 := g_tyBuffer2MagRemoved;
		bRequestToBring3 := g_tyBuffer3MagRemoved;
		//	bRequestToBring4 := g_tyBuffer4MagRemoved;

		bRequestToGet1 := g_tyDSSOT1DBA;
		bRequestToGet2 := g_tyDSSOT2DBA;
		bRequestToGet3 := g_tyDSSOT3DBA;
		//	bRequestToGet4 := g_tyDSSOT4DBA;

		//DMCRFID
		bScanTrigSig := g_tyOpsTravLifStartScanSig;
		bMag1ExitPCB := g_tyOpsTravLifMag1TransOut;
		bMag2ExitPCB := g_tyOpsTravLifMag2TransOut;
		bMag3ExitPCB := g_tyOpsTravLifMag3TransOut;
	ELSE
		bSOTMagReady1 := FALSE;
		bSOTMagReady2 := FALSE;
		bSOTMagReady3 := FALSE;

		bSOTMagError1 := g_tyAlarmErr;
		bSOTMagError2 := g_tyAlarmErr;
		bSOTMagError3 := g_tyAlarmErr;

		bSOTMagAvailable1 := FALSE;
		bSOTMagAvailable2 := FALSE;
		bSOTMagAvailable3 := FALSE;

		bSOTMagSizeLarge1 := FALSE;
		bSOTMagSizeLarge2 := FALSE;
		bSOTMagSizeLarge3 := FALSE;

//		bRequestToBring1 := FALSE;
//		bRequestToBring2 := FALSE;
//		bRequestToBring3 := FALSE;

		bRequestToGet1 := FALSE;
		bRequestToGet2 := FALSE;
		bRequestToGet3 := FALSE;

		//DMCRFID
		bScanTrigSig ACCESS ADR(bStartScanSig);
		bMag1ExitPCB ACCESS ADR(bPCBExitMag1);
		bMag2ExitPCB ACCESS ADR(bPCBExitMag2);
		bMag3ExitPCB ACCESS ADR(bPCBExitMag3);

	END_IF

	CASE p_eLinkAGVComProtocol OF
		McSetAGVCommOPCUA, McSetAGVCommDisabled:
			IF bLinkNtParamProjSOTSenPrep THEN
				bAgvComIODisabled := FALSE;
			ELSE
				bAgvComIODisabled := TRUE;
			END_IF

		McSetAGVCommHardIO:
			bAgvComIODisabled := FALSE;

	END_CASE

	IF g_tyUIOut.bManualMod THEN
		bBypCurtainSen := g_tyUIOut.bMnlBypCurtainSen;
		bRstCurtainSen := g_tyUIOut.bSafetyCurtainReset;
		bBypCurtainPBLED := g_tyUIOut.bMnlBypCurtainPBLED;

	ELSIF g_tyOps.bRun THEN

		bBypCurtainPBLED	 := g_tyOpsTravLifUL.bBypCurtainSensorPBLED;

		IF g_tyOpsTravLifUL.bBypCurtainSenCtrl OR bLinkAGVCommRdy1 OR bLinkAGVCommRdy2 OR bLinkAGVCommRdy3 THEN
			bBypCurtainSen     := TRUE;
		ELSE
			bBypCurtainSen	 := FALSE;
		END_IF

	ELSE
		bRstCurtainSen := g_tyUISafetyCurtainReset;
		bBypCurtainSen := g_tyUIMnlBypCurtainSen;//:= FALSE;
		bBypCurtainPBLED := g_tyUIMnlBypCurtainPBLED;//:= FALSE;
	END_IF

END_ACTION
```

#### Act_InitLocal.st - Change By Project
```iecst
(** 2019-03-25 **)
ACTION Act_InitLocal:

	//Input Reference Link To Local Variable
	p_udiMax ACCESS ADR(c_udiDOutputMax);
	p_eAct ACCESS ADR(eAct);
	p_tyDOSettings ACCESS ADR(tyDOSettings);
	p_bManual ACCESS ADR(bManual);

	p_bSafetyRlyRst ACCESS ADR(bSafetyRlyRst);
	p_bTLRed ACCESS ADR(bTLRed);
	p_bTLAmber ACCESS ADR(bTLAmber);
	p_bTLGreen ACCESS ADR(bTLGreen);
	p_bBuzzer ACCESS ADR(bBuzzer);
	p_bUSBA ACCESS ADR(bUSBA);
	p_bUSBB ACCESS ADR(bUSBB);
	p_bOvenInfoSigA ACCESS ADR(bOvenInfoSigA);
	p_bOvenInfoSigB ACCESS ADR(bOvenInfoSigB);
	p_bPusherExtCtrl ACCESS ADR(bPusherExtCtrl);
	p_bStopperUnblkCtrlA ACCESS ADR(bStopperUnblkCtrlA);
	p_bStopperUnblkCtrlB ACCESS ADR(bStopperUnblkCtrlB);
	p_bMag1FixedClampCtrl ACCESS ADR(bMag1FixedClampCtrl);
	p_bMag1RemoteClampCtrl ACCESS ADR(bMag1RemoteClampCtrl);
	p_bMag2FixedClampCtrl ACCESS ADR(bMag2FixedClampCtrl);
	p_bMag2RemoteClampCtrl ACCESS ADR(bMag2RemoteClampCtrl);
	p_bMag3FixedClampCtrl ACCESS ADR(bMag3FixedClampCtrl);
	p_bMag3RemoteClampCtrl ACCESS ADR(bMag3RemoteClampCtrl);
	p_bInShutterOpenCtrl ACCESS ADR(bInShutterOpenCtrl);
	p_bInShutterCloseCtrl ACCESS ADR(bInShutterCloseCtrl);
	p_bOutShutterOpenCtrl ACCESS ADR(bOutShutterOpenCtrl);
	p_bOutShutterCloseCtrl ACCESS ADR(bOutShutterCloseCtrl);
	p_bMag1ConvMtrIn ACCESS ADR(bMag1ConvMtrIn);
	p_bMag1ConvMtrOut ACCESS ADR(bMag1ConvMtrOut);
	p_bMag2ConvMtrIn ACCESS ADR(bMag2ConvMtrIn);
	p_bMag2ConvMtrOut ACCESS ADR(bMag2ConvMtrOut);
	p_bMag3ConvMtrIn ACCESS ADR(bMag3ConvMtrIn);
	p_bMag3ConvMtrOut ACCESS ADR(bMag3ConvMtrOut);
	p_bMag1SelClampCtrl ACCESS ADR(bMag1SelClampCtrl);
	p_bMag2SelClampCtrl ACCESS ADR(bMag2SelClampCtrl);
	p_bMag3SelClampCtrl ACCESS ADR(bMag3SelClampCtrl);
	p_bPushConvMtrOn ACCESS ADR(bPushConvMtrOn);
	p_bMag1SafetyBarRetCtrl ACCESS ADR(bMag1SafetyBarRetCtrl);
	p_bMag2SafetyBarRetCtrl ACCESS ADR(bMag2SafetyBarRetCtrl);
	p_bMag3SafetyBarRetCtrl ACCESS ADR(bMag3SafetyBarRetCtrl);
	p_bMag1WallEngageCtrl ACCESS ADR(bMag1WallEngageCtrl);
	p_bMag2WallEngageCtrl ACCESS ADR(bMag2WallEngageCtrl);
	p_bMag3WallEngageCtrl ACCESS ADR(bMag3WallEngageCtrl);
	p_bSOTMagError1 ACCESS ADR(bSOTMagError1);
	p_bSOTMagError2 ACCESS ADR(bSOTMagError2);
	p_bSOTMagError3 ACCESS ADR(bSOTMagError3);
	p_bSOTMagError4 ACCESS ADR(bSOTMagError4);
	p_bSOTMagReady1 ACCESS ADR(bSOTMagReady1);
	p_bSOTMagReady2 ACCESS ADR(bSOTMagReady2);
	p_bSOTMagReady3 ACCESS ADR(bSOTMagReady3);
	p_bSOTMagReady4 ACCESS ADR(bSOTMagReady4);
	p_bSOTMagAvailable1 ACCESS ADR(bSOTMagAvailable1);
	p_bSOTMagAvailable2 ACCESS ADR(bSOTMagAvailable2);
	p_bSOTMagAvailable3 ACCESS ADR(bSOTMagAvailable3);
	p_bSOTMagAvailable4 ACCESS ADR(bSOTMagAvailable4);
	p_bSOTMagSizeLarge1 ACCESS ADR(bSOTMagSLarge1);
	p_bSOTMagSizeLarge2 ACCESS ADR(bSOTMagSLarge2);
	p_bSOTMagSizeLarge3 ACCESS ADR(bSOTMagSLarge3);
	p_bSOTMagSizeLarge4 ACCESS ADR(bSOTMagSLarge4);
	p_bMagAWOpenLimByp1 ACCESS ADR(bMagAWOpenLimByp1);
	p_bMagAWOpenLimByp2 ACCESS ADR(bMagAWOpenLimByp2);
	p_bMagAWOpenLimByp3 ACCESS ADR(bMagAWOpenLimByp3);
	p_bMagAWOpenLimByp4 ACCESS ADR(bMagAWOpenLimByp4);
	p_bMagAWSmallLimSen1 ACCESS ADR(bMagAWSmallLimSen1);
	p_bMagAWSmallLimSen2 ACCESS ADR(bMagAWSmallLimSen2);
	p_bMagAWSmallLimSen3 ACCESS ADR(bMagAWSmallLimSen3);
	p_bMagAWSmallLimSen4 ACCESS ADR(bMagAWSmallLimSen4);
	p_bRequestToBring1 ACCESS ADR(bRequestToBring1);
	p_bRequestToGet1 ACCESS ADR(bRequestToGet1);
	p_bRequestToBring2 ACCESS ADR(bRequestToBring2);
	p_bRequestToGet2 ACCESS ADR(bRequestToGet2);
	p_bRequestToBring3 ACCESS ADR(bRequestToBring3);
	p_bRequestToGet3 ACCESS ADR(bRequestToGet3);
	p_bRequestToBring4 ACCESS ADR(bRequestToBring4);
	p_bRequestToGet4 ACCESS ADR(bRequestToGet4);

	p_bEntTopStprUnblkCtrl ACCESS ADR(bEntTopStprUnblkCtrl);
	p_bMidTopStprUnblkCtrl ACCESS ADR(bMidTopStprUnblkCtrl);
	p_bExtTopStprUnblkCtrl ACCESS ADR(bExtTopStprUnblkCtrl);
	p_bMidBtmStprUnblkCtrl ACCESS ADR(bMidBtmStprUnblkCtrl);
	p_bExtBtmStprUnblkCtrl ACCESS ADR(bExtBtmStprUnblkCtrl);
	p_bEntTopStprUnblkCtrl2 ACCESS ADR(bEntTopStprUnblkCtrl2);
	p_bMidTopStprUnblkCtrl2 ACCESS ADR(bMidTopStprUnblkCtrl2);
	p_bExtTopStprUnblkCtrl2 ACCESS ADR(bExtTopStprUnblkCtrl2);
	p_bMidBtmStprUnblkCtrl2 ACCESS ADR(bMidBtmStprUnblkCtrl2);
	p_bExtBtmStprUnblkCtrl2 ACCESS ADR(bExtBtmStprUnblkCtrl2);

	p_bInMagConvMtrOn ACCESS ADR(bInMagConvMtrOn);
	p_bOutMagConvMtrOn ACCESS ADR(bOutMagConvMtrOn);
	p_bInMagConv2MtrOn ACCESS ADR(bInMagConv2MtrOn);
	p_bOutMagConv2MtrOn ACCESS ADR(bOutMagConv2MtrOn);
	p_bMtrPwrRly ACCESS ADR(bMtrPwrRly);

	p_bBypCurtainSen ACCESS ADR(bBypCurtainSen);
	p_bRstCurtainSen ACCESS ADR(bRstCurtainSen);
	p_bBypCurtainPBLED	ACCESS ADR(bBypCurtainPBLED);

END_ACTION
```

#### Act_Main.st - Change By Project
```iecst
(** 2019-01-10 **)
ACTION Act_Main:

	IF eStatOld <> eStat THEN
		sStatTxt	:= a_sStatText[eStat];

		eStatOld	:= eStat;

		eStatus		:= Busy;
	END_IF

	//Main
	CASE eStat OF

		DOActIdle:
			eStatus	:= Idle;

		DOActRstAll:
			IF eStatus = Idle OR eStatus = Busy THEN
				//Sample
//				p_bBypassCoverSwitch	:= FALSE;
				eStatus					:= Done;

			END_IF

		DOActSetBypassCoverSwitch:
			IF eStatus = Idle OR eStatus = Busy THEN
				//Sample
//				p_bBypassCoverSwitch	:= TRUE;
				eStatus					:= Done;

			END_IF

		DOActRstBypassCoverSwitch:
			IF eStatus = Idle OR eStatus = Busy THEN
				//Sample
//				p_bBypassCoverSwitch	:= FALSE;
				eStatus					:= Done;

			END_IF

	END_CASE

END_ACTION
```
